// POUs/Controller/Lvl1/OVN (Oven)/FB_OVN
FUNCTION_BLOCK FB_OVN EXTENDS FB_CtrlBase
VAR_INPUT
	/// 0 = Busy, 1 = OFF, 2 = BeltOn, 3 = Manual, 4 = Run, 5 = Error, 6 = Bundverschlusserkennung 
	In_iStatus: INT;
	/// Machine off 
	In_bOff: BOOL;
	/// Band on 
	In_bBeltOn: BOOL;
	/// Manual 
	In_bManual: BOOL;
	/// Standart drying process 
	In_bRun: BOOL;
	/// Resetting error 
	In_bAckError: BOOL;
	/// Actual temperature in deci °C 
	In_adiTemp_dc: ARRAY[0..(MAX_NUMBER_OF_OVEN_MODULES - 1)] OF DINT;
	/// Aactual airflow in % 
	In_adiAir_p: ARRAY[0..(MAX_NUMBER_OF_OVEN_MODULES - 1)] OF DINT;
	/// Actual belt speed in mm/min 
	In_diSpeed_mm_min: DINT;
	/// 1=Information, 2=Warning, 3=Error 
	In_iErrorLevel: INT;
	/// Error ID (e.g. 100=temperature overflow) 
	In_iErrorID: INT;
	In_bDriverConnected: BOOL;
	In_bDriverError: BOOL;
	In_udiDriverErrorID: UDINT;
	In_uliBarcodeNew_1: ULINT;
	In_uliBarcodeNew_2: ULINT;
	In_uiNewElement_1: UINT;
	In_uiNewElement_2: UINT;
	In_uliBarcodeDelete_1: ULINT;
	In_uliBarcodeDelete_2: ULINT;
	In_uiDeleteElement_1: UINT;
	In_uiDeleteElement_2: UINT;
END_VAR
VAR
	/// Specific interface struct for public access
	SIf: T_Ctrl_SIf_OVN;
	/// this allows to detect parameter changes
	lastSifPar: T_Ctrl_SIf_OVN_Par;
	/// pointer to function block
	p_fbIBH: POINTER TO FB_IBH;
	p_fbIBH_CIf: POINTER TO BASE_PLC.T_Ctrl_CIf;
	/// Monitors
	afbTempMonitors: ARRAY[0..(MAX_NUMBER_OF_OVEN_MODULES - 1)] OF FB_MONITOR;
	afbAirMonitors: ARRAY[0..(MAX_NUMBER_OF_OVEN_MODULES - 1)] OF FB_MONITOR;
	fbSpeedMonitor: FB_MONITOR;
	udiTimeInBand: UDINT;
	/// Tracker
	fbTracker: FB_Tracker;
	/// Error Tracking
	iLastCalledAlarmNr: INT;
	uiNewElementOld_1: UINT;
	uiNewElementOld_2: UINT;
	uiDeleteElementOld_1: UINT;
	uiDeleteElementOld_2: UINT;
END_VAR

(*__________________________________________________________________________________________________
¦	
¦	Vistaprint Schweiz GmbH
¦	CH - 8401 Winterthur
¦
¦	www.vistaprint.ch - info@vistaprint.ch
¦___________________________________________________________________________________________________

Function desription:
Oven Controller Implementation

History:
Version		Date			Author		Comment
---------------------------------------------------------------------------------------------------
0.00.1		10.12.2013		BB			Start history
___________________________________________________________________________________________________*)

// check if child pointer valid
IF (me.bolActivate) THEN // cyclic call enabled
	
	IF (CIf.Info.bolInitDone=FALSE) THEN // first cycle -> init
		CtrlInit();
		CIf.Info.bolInitDone := TRUE;
	ELSE
		CycleStartDuty();
		
		Always();
		
		StateMachine();
		
		CycleEndDuty();
	END_IF
	
END_IF;

{attribute 'object_name' := 'Always'}
METHOD PROTECTED Always : BOOL
VAR
	fbOVN: INT;
	bResettable: BOOL;
END_VAR
SUPER^.Always();

// ----------------------------------------------------------------------------------
// cyclic actions outside of statemachine
IF (me.StateMachine.intState<>cSTA_SINGLE_ANSWER) THEN
	
	// copy number of modules to IBH driver
	p_fbIBH^.getCtrlSIf()^.Cfg.uiNumberOfModules := SIf.Cfg.uiNumberOfModules;
	
	// check parameter from GUI
	THIS^.checkParameter();
	
	// write input values directly to SIf.Cur
	SIf.Cur.diSpeed_mm_min := THIS^.In_diSpeed_mm_min;
	SIf.Cur.adiAir_p := THIS^.In_adiAir_p;
	SIf.Cur.adiTemp_dc := THIS^.In_adiTemp_dc;
	
	// remove old elements from Tracker
	IF In_uiDeleteElement_1<>uiDeleteElementOld_1 THEN
		uiDeleteElementOld_1 := In_uiDeleteElement_1;
		fbTracker.deleteElement(In_uliBarcodeDelete_1, SIf.Cfg.bolDataChannelEnable);
	END_IF
	IF In_uiDeleteElement_2<>uiDeleteElementOld_2 THEN
		uiDeleteElementOld_2 := In_uiDeleteElement_2;
		fbTracker.deleteElement(In_uliBarcodeDelete_2, SIf.Cfg.bolDataChannelEnable);
	END_IF
	
	// update Tracker
	fbTracker.update(In_adiTemp_mc:=In_adiTemp_dc, In_diSpeed_mm_min:=In_diSpeed_mm_min,bolSendToSaber:=SIf.Cfg.bolDataChannelEnable);
	
	// add new elements to Tracker
	IF In_uiNewElement_1<>uiNewElementOld_1 THEN
		uiNewElementOld_1 := In_uiNewElement_1;
		fbTracker.addElement(In_uliBarcodeNew_1);
	END_IF
	IF In_uiNewElement_2<>uiNewElementOld_2 THEN
		uiNewElementOld_2 := In_uiNewElement_2;
		fbTracker.addElement(In_uliBarcodeNew_2);
	END_IF
	
	// check errors when higher than PONBusy
	IF (me.StateMachine.intState>=Base_PLC.cSTA_PON) AND (NOT CIf.SwCfg.bolSimulation) THEN
		
		// go to error if Driver connection is lost
		IF 		NOT THIS^.In_bDriverConnected
			AND	me.StateMachine.intState<>Base_PLC.cSTA_ERROR
			AND	me.StateMachine.intState<>Base_PLC.cSTA_ERRORQuit THEN
				pfbAlarmCtrl^.setAlarm(CIf.Info.intCtrlId,INT_TO_UDINT(E_ALM_OVN.ConnectionError),UDINT_TO_DINT(THIS^.In_udiDriverErrorID),ADR(SIf.Alm),E_AlmState.RST,CIf.Job.eMe_ActivAlmClass);
				me.StateMachine.intStateNext := Base_PLC.cSTA_ERROR;
				iLastCalledAlarmNr := E_ALM_OVN.ConnectionError;
		END_IF
		
		// check Tesoma Errors, ErrorLevel 1 (Info) and 2 (Warning) don't exist
		IF THIS^.In_iErrorLevel=3 THEN
			chooseTesomaErrors(bResettable);
			IF 		me.StateMachine.intState<>Base_PLC.cSTA_ERROR
				AND	me.StateMachine.intState<>Base_PLC.cSTA_ERRORQuit
				and me.StateMachine.intStateNext<>Base_PLC.cSTA_ERROR THEN
					me.StateMachine.intStateNext := Base_PLC.cSTA_ERROR;
			END_IF
		END_IF
		
	END_IF
	
END_IF

// ----------------------------------------------------------------------------------
// overrule error always from base -> no EOFF State!! in EOFF go to OFF
IF (me.StateMachine.intStateNext = cSTA_EOFFBusy) THEN
	IF (me.StateMachine.intState = cSTA_OFF) THEN
		me.StateMachine.intStateNext := cSTA_OFF;
	ELSE // stay in OFF
		me.StateMachine.intStateNext := cSTA_OFFBusy;
	END_IF
END_IF
END_METHOD

{attribute 'object_name' := 'checkParameter'}
METHOD checkParameter : BOOL
VAR
	uiIdx: UINT;
END_VAR
// Belt Speed
IF (SIf.Par.diSpeed_mm_min > SIf.Cfg.diMaxSpeed_mm_min) THEN
	pfbAlarmCtrl^.setAlarm(CIf.Info.intCtrlId,INT_TO_UDINT(E_ALM_OVN.ParameterWarning),0,ADR(SIf.Alm),E_AlmState.RST,CIf.Job.eMe_ActivAlmClass);
	SIf.Par.diSpeed_mm_min := SIf.Cfg.diMaxSpeed_mm_min;
ELSIF (SIf.Par.diSpeed_mm_min < SIf.Cfg.diMinSpeed_mm_min) THEN
	pfbAlarmCtrl^.setAlarm(CIf.Info.intCtrlId,INT_TO_UDINT(E_ALM_OVN.ParameterWarning),0,ADR(SIf.Alm),E_AlmState.RST,CIf.Job.eMe_ActivAlmClass);
	SIf.Par.diSpeed_mm_min := SIf.Cfg.diMinSpeed_mm_min;
END_IF

// Temperature
FOR uiIdx:=0 TO SIf.Cfg.uiNumberOfModules-1 BY 1 DO
	IF (SIf.Par.adiTemp_dc[uiIdx] > SIf.Cfg.diMaxTemp_dc) THEN
		pfbAlarmCtrl^.setAlarm(CIf.Info.intCtrlId,INT_TO_UDINT(E_ALM_OVN.ParameterWarning),uiIdx,ADR(SIf.Alm),E_AlmState.RST,CIf.Job.eMe_ActivAlmClass);
		SIf.Par.adiTemp_dc[uiIdx] := SIf.Cfg.diMaxTemp_dc;
	ELSIF (SIf.Par.adiTemp_dc[uiIdx] < SIf.Cfg.diMinTemp_dc) THEN
		pfbAlarmCtrl^.setAlarm(CIf.Info.intCtrlId,INT_TO_UDINT(E_ALM_OVN.ParameterWarning),uiIdx,ADR(SIf.Alm),E_AlmState.RST,CIf.Job.eMe_ActivAlmClass);
		SIf.Par.adiTemp_dc[uiIdx] := SIf.Cfg.diMinTemp_dc;
	END_IF
END_FOR

// Airflow
FOR uiIdx:=0 TO SIf.Cfg.uiNumberOfModules-1 BY 1 DO
	IF (SIf.Par.adiAir_p[uiIdx] > SIf.Cfg.diMaxAir_p) THEN
		pfbAlarmCtrl^.setAlarm(CIf.Info.intCtrlId,INT_TO_UDINT(E_ALM_OVN.ParameterWarning),uiIdx,ADR(SIf.Alm),E_AlmState.RST,CIf.Job.eMe_ActivAlmClass);
		SIf.Par.adiAir_p[uiIdx] := SIf.Cfg.diMaxAir_p;
	ELSIF (SIf.Par.adiAir_p[uiIdx] < SIf.Cfg.diMinAir_p) THEN
		pfbAlarmCtrl^.setAlarm(CIf.Info.intCtrlId,INT_TO_UDINT(E_ALM_OVN.ParameterWarning),uiIdx,ADR(SIf.Alm),E_AlmState.RST,CIf.Job.eMe_ActivAlmClass);
		SIf.Par.adiAir_p[uiIdx] := SIf.Cfg.diMinAir_p;
	END_IF
END_FOR
END_METHOD

{attribute 'object_name' := 'chooseTesomaErrors'}
METHOD chooseTesomaErrors : BOOL
VAR_IN_OUT
	bResettable: BOOL;
END_VAR
bResettable := FALSE;

CASE THIS^.In_iErrorID OF
	// Tesoma10000
	10000:
		bResettable := TRUE;
		pfbAlarmCtrl^.setAlarm(CIf.Info.intCtrlId,INT_TO_UDINT(E_ALM_OVN.Tesoma10000),In_iErrorID,ADR(SIf.Alm),E_AlmState.RST,CIf.Job.eMe_ActivAlmClass);
	// Tesoma10002
	10002:
		pfbAlarmCtrl^.setAlarm(CIf.Info.intCtrlId,INT_TO_UDINT(E_ALM_OVN.Tesoma10002),In_iErrorID,ADR(SIf.Alm),E_AlmState.RST,CIf.Job.eMe_ActivAlmClass);
	// Tesoma10003
	10003:
		pfbAlarmCtrl^.setAlarm(CIf.Info.intCtrlId,INT_TO_UDINT(E_ALM_OVN.Tesoma10003),In_iErrorID,ADR(SIf.Alm),E_AlmState.RST,CIf.Job.eMe_ActivAlmClass);
	// Tesoma10006
	10006:
		pfbAlarmCtrl^.setAlarm(CIf.Info.intCtrlId,INT_TO_UDINT(E_ALM_OVN.Tesoma10006),In_iErrorID,ADR(SIf.Alm),E_AlmState.RST,CIf.Job.eMe_ActivAlmClass);
	// Tesoma10010
	10010:
		bResettable := TRUE;
		pfbAlarmCtrl^.setAlarm(CIf.Info.intCtrlId,INT_TO_UDINT(E_ALM_OVN.Tesoma10010),In_iErrorID,ADR(SIf.Alm),E_AlmState.RST,CIf.Job.eMe_ActivAlmClass);
	// Tesoma10011
	10011:
		bResettable := TRUE;
		pfbAlarmCtrl^.setAlarm(CIf.Info.intCtrlId,INT_TO_UDINT(E_ALM_OVN.Tesoma10011),In_iErrorID,ADR(SIf.Alm),E_AlmState.RST,CIf.Job.eMe_ActivAlmClass);
	// Tesoma10012
	10012:
		bResettable := TRUE;
		pfbAlarmCtrl^.setAlarm(CIf.Info.intCtrlId,INT_TO_UDINT(E_ALM_OVN.Tesoma10012),In_iErrorID,ADR(SIf.Alm),E_AlmState.RST,CIf.Job.eMe_ActivAlmClass);
	// Tesoma10013
	10013:
		pfbAlarmCtrl^.setAlarm(CIf.Info.intCtrlId,INT_TO_UDINT(E_ALM_OVN.Tesoma10013),In_iErrorID,ADR(SIf.Alm),E_AlmState.RST,CIf.Job.eMe_ActivAlmClass);
	// Tesoma10014
	10014:
		bResettable := TRUE;
		pfbAlarmCtrl^.setAlarm(CIf.Info.intCtrlId,INT_TO_UDINT(E_ALM_OVN.Tesoma10014),In_iErrorID,ADR(SIf.Alm),E_AlmState.RST,CIf.Job.eMe_ActivAlmClass);
	// Tesoma10016
	10016:
		pfbAlarmCtrl^.setAlarm(CIf.Info.intCtrlId,INT_TO_UDINT(E_ALM_OVN.Tesoma10016),In_iErrorID,ADR(SIf.Alm),E_AlmState.RST,CIf.Job.eMe_ActivAlmClass);
	// Tesoma10023
	10023:
		pfbAlarmCtrl^.setAlarm(CIf.Info.intCtrlId,INT_TO_UDINT(E_ALM_OVN.Tesoma10023),In_iErrorID,ADR(SIf.Alm),E_AlmState.RST,CIf.Job.eMe_ActivAlmClass);
	// Tesoma10024
	10024:
		pfbAlarmCtrl^.setAlarm(CIf.Info.intCtrlId,INT_TO_UDINT(E_ALM_OVN.Tesoma10024),In_iErrorID,ADR(SIf.Alm),E_AlmState.RST,CIf.Job.eMe_ActivAlmClass);
	// Tesoma10025
	10025:
		pfbAlarmCtrl^.setAlarm(CIf.Info.intCtrlId,INT_TO_UDINT(E_ALM_OVN.Tesoma10025),In_iErrorID,ADR(SIf.Alm),E_AlmState.RST,CIf.Job.eMe_ActivAlmClass);
	// Tesoma10026
	10026:
		pfbAlarmCtrl^.setAlarm(CIf.Info.intCtrlId,INT_TO_UDINT(E_ALM_OVN.Tesoma10026),In_iErrorID,ADR(SIf.Alm),E_AlmState.RST,CIf.Job.eMe_ActivAlmClass);
	// Tesoma10027
	10027:
		pfbAlarmCtrl^.setAlarm(CIf.Info.intCtrlId,INT_TO_UDINT(E_ALM_OVN.Tesoma10027),In_iErrorID,ADR(SIf.Alm),E_AlmState.RST,CIf.Job.eMe_ActivAlmClass);
	// Tesoma10030
	10030:
		pfbAlarmCtrl^.setAlarm(CIf.Info.intCtrlId,INT_TO_UDINT(E_ALM_OVN.Tesoma10030),In_iErrorID,ADR(SIf.Alm),E_AlmState.RST,CIf.Job.eMe_ActivAlmClass);
	// Tesoma10031
	10031:
		pfbAlarmCtrl^.setAlarm(CIf.Info.intCtrlId,INT_TO_UDINT(E_ALM_OVN.Tesoma10031),In_iErrorID,ADR(SIf.Alm),E_AlmState.RST,CIf.Job.eMe_ActivAlmClass);
	// Tesoma10032
	10032:
		pfbAlarmCtrl^.setAlarm(CIf.Info.intCtrlId,INT_TO_UDINT(E_ALM_OVN.Tesoma10032),In_iErrorID,ADR(SIf.Alm),E_AlmState.RST,CIf.Job.eMe_ActivAlmClass);
	// Tesoma10034
	10034:
		pfbAlarmCtrl^.setAlarm(CIf.Info.intCtrlId,INT_TO_UDINT(E_ALM_OVN.Tesoma10034),In_iErrorID,ADR(SIf.Alm),E_AlmState.RST,CIf.Job.eMe_ActivAlmClass);
	// Tesoma10x00
	10100, 10200, 10300, 10400, 10500, 10600, 10700, 10800, 10900:
		bResettable := TRUE;
		pfbAlarmCtrl^.setAlarm(CIf.Info.intCtrlId,INT_TO_UDINT(E_ALM_OVN.Tesoma10x00),In_iErrorID,ADR(SIf.Alm),E_AlmState.RST,CIf.Job.eMe_ActivAlmClass);
	// Tesoma10x01
	10101, 10201, 10301, 10401, 10501, 10601, 10701, 10801, 10901:
		bResettable := TRUE;
		pfbAlarmCtrl^.setAlarm(CIf.Info.intCtrlId,INT_TO_UDINT(E_ALM_OVN.Tesoma10x01),In_iErrorID,ADR(SIf.Alm),E_AlmState.RST,CIf.Job.eMe_ActivAlmClass);
	// Tesoma10x02
	10102, 10202, 10302, 10402, 10502, 10602, 10702, 10802, 10902:
		bResettable := TRUE;
		pfbAlarmCtrl^.setAlarm(CIf.Info.intCtrlId,INT_TO_UDINT(E_ALM_OVN.Tesoma10x02),In_iErrorID,ADR(SIf.Alm),E_AlmState.RST,CIf.Job.eMe_ActivAlmClass);
	// Tesoma10x03
	10103, 10203, 10303, 10403, 10503, 10603, 10703, 10803, 10903:
		bResettable := TRUE;
		pfbAlarmCtrl^.setAlarm(CIf.Info.intCtrlId,INT_TO_UDINT(E_ALM_OVN.Tesoma10x03),In_iErrorID,ADR(SIf.Alm),E_AlmState.RST,CIf.Job.eMe_ActivAlmClass);
	// Tesoma10x07
	10107, 10207, 10307, 10407, 10507, 10607, 10707, 10807, 10907:
		bResettable := TRUE;
		pfbAlarmCtrl^.setAlarm(CIf.Info.intCtrlId,INT_TO_UDINT(E_ALM_OVN.Tesoma10x07),In_iErrorID,ADR(SIf.Alm),E_AlmState.RST,CIf.Job.eMe_ActivAlmClass);
	// Tesoma10x13
	10113, 10213, 10313, 10413, 10513, 10613, 10713, 10813, 10913:
		pfbAlarmCtrl^.setAlarm(CIf.Info.intCtrlId,INT_TO_UDINT(E_ALM_OVN.Tesoma10x13),In_iErrorID,ADR(SIf.Alm),E_AlmState.RST,CIf.Job.eMe_ActivAlmClass);
	// Tesoma10x14
	10114, 10214, 10314, 10414, 10514, 10614, 10714, 10814, 10914:
		pfbAlarmCtrl^.setAlarm(CIf.Info.intCtrlId,INT_TO_UDINT(E_ALM_OVN.Tesoma10x14),In_iErrorID,ADR(SIf.Alm),E_AlmState.RST,CIf.Job.eMe_ActivAlmClass);
	// Tesoma10x15
	10115, 10215, 10315, 10415, 10515, 10615, 10715, 10815, 10915:
		pfbAlarmCtrl^.setAlarm(CIf.Info.intCtrlId,INT_TO_UDINT(E_ALM_OVN.Tesoma10x15),In_iErrorID,ADR(SIf.Alm),E_AlmState.RST,CIf.Job.eMe_ActivAlmClass);
	// Tesoma13x00
	13100, 13200, 13300, 13400, 13500, 13600, 13700, 13800, 13900:
		bResettable := TRUE;
		pfbAlarmCtrl^.setAlarm(CIf.Info.intCtrlId,INT_TO_UDINT(E_ALM_OVN.Tesoma13x00),In_iErrorID,ADR(SIf.Alm),E_AlmState.RST,CIf.Job.eMe_ActivAlmClass);
ELSE
	// TesomaUnknown
		pfbAlarmCtrl^.setAlarm(CIf.Info.intCtrlId,INT_TO_UDINT(E_ALM_OVN.TesomaUnknown),In_iErrorID,ADR(SIf.Alm),E_AlmState.RST,CIf.Job.eMe_ActivAlmClass);
END_CASE
END_METHOD

{attribute 'object_name' := 'CtrlInit'}
METHOD CtrlInit : BOOL
SUPER^.CtrlInit();

// add childs
p_fbIBH_CIf := THIS^.AddChild(p_fbIBH^);

// Tracker Init
fbTracker.numberOfModules := SIf.Cfg.uiNumberOfModules;
fbTracker.sampleTime_us := me.FUBInfo.udiSample_us;
fbTracker.moduleLength_mm := SIf.Cfg.diModuleLength_mm;
fbTracker.distanceBeforeOven_mm := SIf.Cfg.diDistanceBeforeOven_mm;	//TODO: BB: This should be the distance from the barcode reader to the begin of the first module of the oven
fbTracker.distanceAfterOven_mm := SIf.Cfg.diDistanceAfterOven_mm;	//TODO: BB: This should be the distance from the barcode reader to the end of the first module of the oven
END_METHOD

PROPERTY PUBLIC CtrlSIf : POINTER TO T_Ctrl_SIf_OVN
GET
CtrlSIf := ADR(SIf);
END_GET
END_PROPERTY

PROPERTY DataChannel : POINTER TO FB_DataChannelSenderFifo
SET
fbTracker.DataChannel := DataChannel;
END_SET
END_PROPERTY

{attribute 'object_name' := 'FB_init'}
METHOD FB_init : BOOL
VAR_INPUT
	///if TRUE, the retain variables are initialized (warm start / cold start)
	bInitRetains: BOOL;
	///if TRUE, the instance afterwards gets moved into the copy code (online change)
	bInCopyCode: BOOL;
END_VAR
VAR
	uiIdx: UINT;
END_VAR
//------------------------------------------------------------------------------------------------------------------------
// to manually change in new FUB implementation!!!
// define valid commands for this controller
FOR uiIdx:=0 TO (SIZEOF(CIf.Job.aCmdList)/SIZEOF(CIf.Job.aCmdList[0])-1) BY 1 DO
	IF (CIf.Job.aCmdList[uiIdx].intCmd=cSTA_INITIALIZED) THEN
		// found first empty array element
		EXIT;
	END_IF
END_FOR

// Add configuration of own comands
CIf.Job.aCmdList[uiIdx].intCmd := OVN_CmdState.cCMD_BELTONLY;
CIf.Job.aCmdList[uiIdx].strName := 'BELTONLY';
CIf.Job.aCmdList[uiIdx].bolAvailable := TRUE;
uiIdx := uiIdx+1;
CIf.Job.aCmdList[uiIdx].intCmd := Base_PLC.cCMD_RUN;
CIf.Job.aCmdList[uiIdx].strName := 'RUN';
CIf.Job.aCmdList[uiIdx].bolAvailable := TRUE;

// set name of class/typ
CIf.Info.strType := 'FB_OVN';
CIf.Info.strFullName := 'Oven';

// set alarm class
SIf.Alm[E_ALM_OVN.TempError].eAlmClass := E_AlmClass.TSTOP;
SIf.Alm[E_ALM_OVN.TempError].strText := 'Temperature Error';
SIf.Alm[E_ALM_OVN.AirError].eAlmClass := E_AlmClass.TSTOP;
SIf.Alm[E_ALM_OVN.AirError].strText := 'Airflow Error';
SIf.Alm[E_ALM_OVN.SpeedError].eAlmClass := E_AlmClass.TSTOP;
SIf.Alm[E_ALM_OVN.SpeedError].strText := 'Band Speed Error';
SIf.Alm[E_ALM_OVN.TimeoutError].eAlmClass := E_AlmClass.TSTOP;
SIf.Alm[E_ALM_OVN.TimeoutError].strText := 'Timeout Error on State Change';
SIf.Alm[E_ALM_OVN.ParameterWarning].eAlmClass := E_AlmClass.WARNING;
SIf.Alm[E_ALM_OVN.ParameterWarning].strText := 'Parameter Warning - Parameters got adjusted within the allowed limits';
SIf.Alm[E_ALM_OVN.ConnectionError].eAlmClass := E_AlmClass.TSTOP;
SIf.Alm[E_ALM_OVN.ConnectionError].strText := 'Connection Error';
SIf.Alm[E_ALM_OVN.WrongMode].eAlmClass := E_AlmClass.TSTOP;
SIf.Alm[E_ALM_OVN.WrongMode].strText := 'Wrong Mode - Possible Manual Intervention';

SIf.Alm[E_ALM_OVN.Tesoma10000].eAlmClass := E_AlmClass.TSTOP;
SIf.Alm[E_ALM_OVN.Tesoma10000].strText := 'Tesoma - Overtemperature Power Section';
SIf.Alm[E_ALM_OVN.Tesoma10002].eAlmClass := E_AlmClass.TSTOP;
SIf.Alm[E_ALM_OVN.Tesoma10002].strText := 'Tesoma - Failure of Active Cooling Unit';
SIf.Alm[E_ALM_OVN.Tesoma10003].eAlmClass := E_AlmClass.TSTOP;
SIf.Alm[E_ALM_OVN.Tesoma10003].strText := 'Tesoma - Active Cooling Unit not Running';
SIf.Alm[E_ALM_OVN.Tesoma10006].eAlmClass := E_AlmClass.TSTOP;
SIf.Alm[E_ALM_OVN.Tesoma10006].strText := 'Tesoma - Failure Fuse General';
SIf.Alm[E_ALM_OVN.Tesoma10010].eAlmClass := E_AlmClass.TSTOP;
SIf.Alm[E_ALM_OVN.Tesoma10010].strText := 'Tesoma - Belt Position Control Sensor Error';
SIf.Alm[E_ALM_OVN.Tesoma10011].eAlmClass := E_AlmClass.TSTOP;
SIf.Alm[E_ALM_OVN.Tesoma10011].strText := 'Tesoma - Belt Edge Shut Off';
SIf.Alm[E_ALM_OVN.Tesoma10012].eAlmClass := E_AlmClass.TSTOP;
SIf.Alm[E_ALM_OVN.Tesoma10012].strText := 'Tesoma - Fault Belt Speed';
SIf.Alm[E_ALM_OVN.Tesoma10013].eAlmClass := E_AlmClass.TSTOP;
SIf.Alm[E_ALM_OVN.Tesoma10013].strText := 'Tesoma - Transport Overload';
SIf.Alm[E_ALM_OVN.Tesoma10014].eAlmClass := E_AlmClass.TSTOP;
SIf.Alm[E_ALM_OVN.Tesoma10014].strText := 'Tesoma - Belt Control Device Fault';
SIf.Alm[E_ALM_OVN.Tesoma10016].eAlmClass := E_AlmClass.TSTOP;
SIf.Alm[E_ALM_OVN.Tesoma10016].strText := 'Tesoma - Emergency Stop';
SIf.Alm[E_ALM_OVN.Tesoma10023].eAlmClass := E_AlmClass.TSTOP;
SIf.Alm[E_ALM_OVN.Tesoma10023].strText := 'Tesoma - Belt Wear Monitor';
SIf.Alm[E_ALM_OVN.Tesoma10024].eAlmClass := E_AlmClass.TSTOP;
SIf.Alm[E_ALM_OVN.Tesoma10024].strText := 'Tesoma - Control Cabinet Fan';
SIf.Alm[E_ALM_OVN.Tesoma10025].eAlmClass := E_AlmClass.TSTOP;
SIf.Alm[E_ALM_OVN.Tesoma10025].strText := 'Tesoma - Control Cabinet Temperature too High';
SIf.Alm[E_ALM_OVN.Tesoma10026].eAlmClass := E_AlmClass.TSTOP;
SIf.Alm[E_ALM_OVN.Tesoma10026].strText := 'Tesoma - Power Supply Failure';
SIf.Alm[E_ALM_OVN.Tesoma10027].eAlmClass := E_AlmClass.TSTOP;
SIf.Alm[E_ALM_OVN.Tesoma10027].strText := 'Tesoma - Intake Hood Temperature Exceeded';
SIf.Alm[E_ALM_OVN.Tesoma10030].eAlmClass := E_AlmClass.TSTOP;
SIf.Alm[E_ALM_OVN.Tesoma10030].strText := 'Tesoma - Air Pressure too low';
SIf.Alm[E_ALM_OVN.Tesoma10031].eAlmClass := E_AlmClass.TSTOP;
SIf.Alm[E_ALM_OVN.Tesoma10031].strText := 'Tesoma - Belt Position Control not Working';
SIf.Alm[E_ALM_OVN.Tesoma10032].eAlmClass := E_AlmClass.TSTOP;
SIf.Alm[E_ALM_OVN.Tesoma10032].strText := 'Tesoma - Error Cooling Device Control Cabinet';
SIf.Alm[E_ALM_OVN.Tesoma10034].eAlmClass := E_AlmClass.TSTOP;
SIf.Alm[E_ALM_OVN.Tesoma10034].strText := 'Tesoma - Control Cabinet Cooler and Small Drives Fuse Failure';
SIf.Alm[E_ALM_OVN.Tesoma10x00].eAlmClass := E_AlmClass.TSTOP;
SIf.Alm[E_ALM_OVN.Tesoma10x00].strText := 'Tesoma - LimitSwitchingOff';
SIf.Alm[E_ALM_OVN.Tesoma10x01].eAlmClass := E_AlmClass.TSTOP;
SIf.Alm[E_ALM_OVN.Tesoma10x01].strText := 'Tesoma - Overtemperature Safety Temperature Limiter';
SIf.Alm[E_ALM_OVN.Tesoma10x02].eAlmClass := E_AlmClass.TSTOP;
SIf.Alm[E_ALM_OVN.Tesoma10x02].strText := 'Tesoma - Fuse Triggered';
SIf.Alm[E_ALM_OVN.Tesoma10x03].eAlmClass := E_AlmClass.TSTOP;
SIf.Alm[E_ALM_OVN.Tesoma10x03].strText := 'Tesoma - Failure Exhaust Air Differential Pressure Sensor';
SIf.Alm[E_ALM_OVN.Tesoma10x07].eAlmClass := E_AlmClass.TSTOP;
SIf.Alm[E_ALM_OVN.Tesoma10x07].strText := 'Tesoma - Error Frequency Converter';
SIf.Alm[E_ALM_OVN.Tesoma10x13].eAlmClass := E_AlmClass.TSTOP;
SIf.Alm[E_ALM_OVN.Tesoma10x13].strText := 'Tesoma - Temperature Sensor IR Defective';
SIf.Alm[E_ALM_OVN.Tesoma10x14].eAlmClass := E_AlmClass.TSTOP;
SIf.Alm[E_ALM_OVN.Tesoma10x14].strText := 'Tesoma - Fault Frame Cooling System Differential Pressure Sensor';
SIf.Alm[E_ALM_OVN.Tesoma10x15].eAlmClass := E_AlmClass.TSTOP;
SIf.Alm[E_ALM_OVN.Tesoma10x15].strText := 'Tesoma - Fault Exhaust Air Differential Pressure Sensor';
SIf.Alm[E_ALM_OVN.Tesoma13x00].eAlmClass := E_AlmClass.TSTOP;
SIf.Alm[E_ALM_OVN.Tesoma13x00].strText := 'Tesoma - Temperature Fault';
SIf.Alm[E_ALM_OVN.TesomaUnknown].eAlmClass := E_AlmClass.TSTOP;
SIf.Alm[E_ALM_OVN.TesomaUnknown].strText := 'Tesoma - Unknown Error';
SIf.Alm[E_ALM_OVN.HostConnectionLost].eAlmClass := E_AlmClass.TSTOP;
SIf.Alm[E_ALM_OVN.HostConnectionLost].strText := 'Saber Communication Lost';
SIf.Alm[E_ALM_OVN.SettingsChanged].eAlmClass := E_AlmClass.TSTOP;
SIf.Alm[E_ALM_OVN.SettingsChanged].strText := 'Settings Changed';

//*******************************************************************************
// initial values
//*******************************************************************************

// Software configuration
CIf.SwCfg.bolExist := TRUE;
CIf.SwCfg.bolEnable := TRUE;
CIf.SwCfg.bolSimulation := FALSE;

// Configuration
SIf.Cfg.uiNumberOfModules := 4;
SIf.Cfg.diModuleLength_mm := 2000;
SIf.Cfg.diDistanceBeforeOven_mm := 1000;
SIf.Cfg.diDistanceAfterOven_mm := 1000;
SIf.Cfg.diMinAir_p := 40;
SIf.Cfg.diMaxAir_p := 100;
SIf.Cfg.diMaxSpeed_mm_min := 30000;
SIf.Cfg.diMinSpeed_mm_min := 3000;
SIf.Cfg.diMinTemp_dc := 0;
SIf.Cfg.diMaxTemp_dc := 2000;
SIf.Cfg.bAutoContinueAfterConnectionError := FALSE;
SIf.Cfg.bolDataChannelEnable := FALSE;
SIf.Cfg.bIgnoreOffBusyWaitPaper := FALSE;

// Parameter
SIf.Par.diSpeed_mm_min := SIf.Cfg.diMinSpeed_mm_min;
SIf.Par.diSpeedBand1_mm_min := 100;
SIf.Par.diSpeedBand2_mm_min := 200;
SIf.Par.udiSpeedTimeout_ms := 5000;
SIf.Par.udiTimeoutOffBusy_ms := 2000;
SIf.Par.udiTimeoutRunBusyReaction_ms := 1000;
SIf.Par.udiTimeoutRunBusyInBand_ms := 1*60*1000;
SIf.Par.udiTimeoutBeltOnlyReaction_ms := 1000;
SIf.Par.udiTimeoutBeltOnlyBusy_ms := 10000;

FOR uiIdx:=0 TO MAX_NUMBER_OF_OVEN_MODULES-1 BY 1 DO
	SIf.Par.adiTemp_dc[uiIdx] := 1000;
	SIf.Par.adiTempBand1_dc[uiIdx] := 30;
	SIf.Par.adiTempBand2_dc[uiIdx] := 60;
	SIf.Par.audiTempTimeout_ms[uiIdx] := 5000;
	SIf.Par.adiAir_p[uiIdx] := SIf.Cfg.diMinAir_p;
	SIf.Par.adiAirBand1_p[uiIdx] := 2;
	SIf.Par.adiAirBand2_p[uiIdx] := 4;
	SIf.Par.audiAirTimeout_ms[uiIdx] := 5000;
END_FOR
END_METHOD

{attribute 'object_name' := 'getCmdState'}
METHOD PROTECTED getCmdState : STRING
VAR_INPUT
	intCmdState: INT;
	bolState: BOOL;
END_VAR
getCmdState := SUPER^.getCmdState(intCmdState:=intCmdState,bolState:=bolState); // get global/base defined cmds/states

IF (getCmdState='') THEN // global not defined get local
	// get string cmd/state string information in runtime
	IF (bolState=FALSE) THEN
		// cmd's
		CASE intCmdState OF
			OVN_CmdState.cCMD_BELTONLY:
				getCmdState := 'BELTONLY';
		ELSE
			getCmdState := 'Cmd not defined';
		END_CASE;
	ELSE
		// state's
		CASE intCmdState OF
			OVN_CmdState.cSTA_BELTONLY: 
				getCmdState := 'BELTONLY';
			OVN_CmdState.cSTA_BELTONLYbusy: 
				getCmdState := 'BELTONLYbusy';
			OVN_CmdState.cSUB_WAITOFF: 
				getCmdState := 'WAITOFF';
			OVN_CmdState.cSUB_WAITPAPER: 
				getCmdState := 'WAITPAPER';
			OVN_CmdState.cSUB_DONE: 
				getCmdState := 'DONE';
		ELSE
			getCmdState := 'State not defined';
		END_CASE;
	END_IF
END_IF
END_METHOD

{attribute 'object_name' := 'getCtrlSIf'}
METHOD getCtrlSIf : POINTER TO T_Ctrl_SIf_OVN
getCtrlSIf := ADR(SIf);
END_METHOD

PROPERTY IBH : POINTER TO FB_IBH
GET
IBH := p_fbIBH;
END_GET
SET
p_fbIBH := IBH;
END_SET
END_PROPERTY

{attribute 'object_name' := 'sta_BELTONLY'}
METHOD PROTECTED sta_BELTONLY : BOOL
VAR
	uiIdx: UINT;
END_VAR
// state implemetation

// Entry action
//--------------------------------------------------------------------------------------
	IF (me.StateMachine.intState <> me.StateMachine.intStateLastCycle) THEN
		// state changed since last cycle
		me.StateMachine.intStateLastCycle := me.StateMachine.intState;
	END_IF

	
// Cyclic action
//--------------------------------------------------------------------------------------

	// check if parameters have changed
	IF (TC2_SYSTEM.MEMCMP(pBuf1:=ADR(SIf.Par), pBuf2:=ADR(THIS^.lastSifPar), n:=SIZEOF(SIf.Par)) <> 0) THEN
		me.StateMachine.intStateNext := OVN_CmdState.cSTA_BELTONLYBusy;
	END_IF
	
	IF NOT In_bBeltOn OR NOT (In_iStatus=2 OR In_iStatus=6 OR In_iStatus=5) THEN
		pfbAlarmCtrl^.setAlarm(CIf.Info.intCtrlId,INT_TO_UDINT(E_ALM_OVN.WrongMode),0,ADR(SIf.Alm),E_AlmState.RST,CIf.Job.eMe_ActivAlmClass);
		me.StateMachine.intStateNext := Base_PLC.cSTA_ERROR;
	END_IF
	
	// State Change Condition
	IF (me.StateMachine.intStateNext <> Base_PLC.cSTA_ERROR) THEN
		CASE me.intCmd OF
			Base_PLC.cCMD_OFF:
				me.StateMachine.intStateNext := Base_PLC.cSTA_OFFBusy;
		END_CASE
	END_IF


// Exit action
//--------------------------------------------------------------------------------------
	IF (me.StateMachine.intState <> me.StateMachine.intStateNext) THEN
		// state is going to change
		;
	END_IF
END_METHOD

{attribute 'object_name' := 'sta_BELTONLYBusy'}
METHOD PROTECTED sta_BELTONLYBusy : BOOL
VAR
	uiIdx: UINT;
	bReady: BOOL;
	iErrorNumber: INT;
END_VAR
// state implemetation

// Entry action
//--------------------------------------------------------------------------------------
	IF (me.StateMachine.intState <> me.StateMachine.intStateLastCycle) THEN
		// state changed since last cycle
		me.StateMachine.intStateLastCycle := me.StateMachine.intState;
		
		// Set Outputs
		p_fbIBH^.setBeltOn();
		p_fbIBH^.setSpeed(In_diSpeed_mm_min := SIf.Par.diSpeed_mm_min);
		THIS^.lastSifPar := SIf.Par;
	END_IF
	
	
// Cyclic action
//--------------------------------------------------------------------------------------
	
	// check if parameters have changed
	IF (TC2_SYSTEM.MEMCMP(pBuf1:=ADR(SIf.Par), pBuf2:=ADR(THIS^.lastSifPar), n:=SIZEOF(SIf.Par)) <> 0) THEN
		p_fbIBH^.setSpeed(In_diSpeed_mm_min := SIf.Par.diSpeed_mm_min);
		THIS^.lastSifPar := SIf.Par;
	END_IF
	
	// check timeouts
	IF me.StateMachine.udiTimeInState_ms>SIf.Par.udiTimeoutBeltOnlyBusy_ms THEN
		iErrorNumber := 100*me.StateMachine.intState+In_iStatus;
		pfbAlarmCtrl^.setAlarm(CIf.Info.intCtrlId,INT_TO_UDINT(E_ALM_OVN.TimeoutError),iErrorNumber,ADR(SIf.Alm),E_AlmState.RST,CIf.Job.eMe_ActivAlmClass);
		me.StateMachine.intStateNext := Base_PLC.cSTA_ERROR;
	ELSIF me.StateMachine.udiTimeInState_ms>SIf.Par.udiTimeoutBeltOnlyReaction_ms THEN
		IF NOT In_bBeltOn OR NOT ((In_iStatus=2) OR (In_iStatus=6)) THEN
			iErrorNumber := 100*me.StateMachine.intState+In_iStatus;
			pfbAlarmCtrl^.setAlarm(CIf.Info.intCtrlId,INT_TO_UDINT(E_ALM_OVN.TimeoutError),iErrorNumber,ADR(SIf.Alm),E_AlmState.RST,CIf.Job.eMe_ActivAlmClass);
			me.StateMachine.intStateNext := Base_PLC.cSTA_ERROR;
		END_IF
	END_IF
	
	// Check if ready
	bReady := TRUE;
	IF NOT In_bBeltOn OR NOT ((In_iStatus=2) OR (In_iStatus=6)) THEN
		bReady := FALSE;
	END_IF
	IF (ABS(THIS^.In_diSpeed_mm_min - SIf.Par.diSpeed_mm_min) > ABS(SIf.Par.diSpeedBand1_mm_min)) THEN
		bReady := FALSE;
	END_IF
	
	// State Change Condition
	IF (me.StateMachine.intStateNext <> Base_PLC.cSTA_ERROR) THEN
		CASE me.intCmd OF
			// OFF
			Base_PLC.cCMD_OFF:
				me.StateMachine.intStateNext := Base_PLC.cSTA_OFFBusy;
		ELSE
			// DEFAULT
			IF bReady THEN
				me.StateMachine.intStateNext := OVN_CmdState.cSTA_BELTONLY;
			END_IF
		END_CASE
	END_IF


// Exit action
//--------------------------------------------------------------------------------------
	IF (me.StateMachine.intState <> me.StateMachine.intStateNext) THEN
		// state is going to change
		;
	END_IF
END_METHOD

{attribute 'object_name' := 'sta_ERROR'}
METHOD PROTECTED sta_ERROR : BOOL
// state implemetation

// Entry action
//--------------------------------------------------------------------------------------
	IF (me.StateMachine.intState <> me.StateMachine.intStateLastCycle) THEN
		// state changed since last cycle
		me.StateMachine.intStateHistory := me.StateMachine.intStateLastCycle; // -> possibillity to go back to state before error
		me.StateMachine.intStateLastCycle := me.StateMachine.intState;
	END_IF

	
// Cyclic action
//--------------------------------------------------------------------------------------	
	
	// Mark all tracked item as trash
	fbTracker.markAllTrash();
	
	// auto continue after Connection Error
	IF (iLastCalledAlarmNr=E_ALM_OVN.ConnectionError AND SIf.Cfg.bAutoContinueAfterConnectionError) THEN
		IF THIS^.In_bDriverConnected THEN
			CIf.Job.bolAlmReset := TRUE;
			pfbAlarmCtrl^.setAlarm(CIf.Info.intCtrlId,INT_TO_UDINT(E_ALM_OVN.ConnectionError),UDINT_TO_DINT(THIS^.In_udiDriverErrorID),ADR(SIf.Alm),E_AlmState.CLR,CIf.Job.eMe_ActivAlmClass);
		END_IF
	END_IF
	
	// State Change Condition
	IF (CIf.Job.bolAlmReset = TRUE) THEN
		IF (p_fbIBH_CIf^.Job.intState = cSTA_OFF) THEN
			// Start Driver
			p_fbIBH_CIf^.Job.intACmd := IBH_CmdState.cCMD_CONNECT;
		END_IF
		p_fbIBH^.setAckError();
		me.StateMachine.intStateNext := cSTA_ERRORQuit;
	END_IF


// Exit action
//--------------------------------------------------------------------------------------
	IF (me.StateMachine.intState <> me.StateMachine.intStateNext) THEN
		// state is going to change
		;
	END_IF
END_METHOD

{attribute 'object_name' := 'sta_ERRORQuit'}
METHOD PROTECTED sta_ERRORQuit : BOOL
// state implemetation

// Entry action
//--------------------------------------------------------------------------------------
	IF (me.StateMachine.intState <> me.StateMachine.intStateLastCycle) THEN
		// state changed since last cycle
		me.StateMachine.intStateLastCycle := me.StateMachine.intState;
	END_IF

	
// Cyclic action
//--------------------------------------------------------------------------------------	
	
	// State Change Condition
	CASE me.StateMachine.intStateHistory OF
		// RUN
		Base_PLC.cSTA_RUN, Base_PLC.cSTA_RUNBusy:
			me.StateMachine.intStateNext := Base_PLC.cSTA_RUNBusy;
		// PON
		Base_PLC.cSTA_PON, Base_PLC.cSTA_PONBusy:
			me.StateMachine.intStateNext := Base_PLC.cSTA_PONBusy;
		// STOP
		Base_PLC.cSTA_STOP, Base_PLC.cSTA_STOPBusy:
			me.StateMachine.intStateNext := Base_PLC.cSTA_STOPBusy;
		// BELTONLY
		OVN_CmdState.cSTA_BELTONLY, OVN_CmdState.cSTA_BELTONLYBusy:
			me.StateMachine.intStateNext := OVN_CmdState.cSTA_BELTONLYBusy;
	ELSE
		// DEFAULT
		me.StateMachine.intStateNext := Base_PLC.cSTA_OFFBusy;
	END_CASE


// Exit action
//--------------------------------------------------------------------------------------
	IF (me.StateMachine.intState <> me.StateMachine.intStateNext) THEN
		// state is going to change
		
		// Reset iLastCalledAlarmNr
		iLastCalledAlarmNr := E_ALM_OVN.NONE;
	END_IF
END_METHOD

{attribute 'object_name' := 'sta_OFF'}
METHOD PROTECTED sta_OFF : BOOL
VAR
	uiIdx: UINT;
END_VAR
// state implemetation

// Entry action
//--------------------------------------------------------------------------------------
	IF (me.StateMachine.intState <> me.StateMachine.intStateLastCycle) THEN
		// state changed since last cycle
		me.StateMachine.intStateLastCycle := me.StateMachine.intState;
	END_IF

	
// Cyclic action
//--------------------------------------------------------------------------------------
	
	IF NOT In_bOff OR NOT (In_iStatus=1 OR In_iStatus=6 OR In_iStatus=5) THEN
		pfbAlarmCtrl^.setAlarm(CIf.Info.intCtrlId,INT_TO_UDINT(E_ALM_OVN.WrongMode),0,ADR(SIf.Alm),E_AlmState.RST,CIf.Job.eMe_ActivAlmClass);
		me.StateMachine.intStateNext := Base_PLC.cSTA_ERROR;
	END_IF
	
	// State Change Condition
	IF (me.StateMachine.intStateNext <> Base_PLC.cSTA_ERROR) THEN
		CASE me.intCmd OF
			// RUN
			Base_PLC.cCMD_RUN:
				me.StateMachine.intStateNext := Base_PLC.cSTA_RUNBusy;
			// BELTONLY
			OVN_CmdState.cCMD_BELTONLY:
				me.StateMachine.intStateNext := OVN_CmdState.cSTA_BELTONLYBusy;
		ELSE
			// DEFAULT
			;
		END_CASE
	END_IF


// Exit action
//--------------------------------------------------------------------------------------
	IF (me.StateMachine.intState <> me.StateMachine.intStateNext) THEN
		// state is going to change
		;
	END_IF
END_METHOD

{attribute 'object_name' := 'sta_OFFBusy'}
METHOD PROTECTED sta_OFFBusy : BOOL
VAR
	bReady: BOOL;
	iErrorNumber: INT;
	uiIdx: UINT;
	udiCoolDownTime_ms: UDINT;
END_VAR
// state implemetation

// Entry action
//--------------------------------------------------------------------------------------
	IF (me.StateMachine.intState <> me.StateMachine.intStateLastCycle) THEN
		// state changed since last cycle
		me.StateMachine.intStateLastCycle := me.StateMachine.intState;
		me.SubStateMachine.intState 	:= OVN_CmdState.cSUB_WAITOFF;
		me.SubStateMachine.intStateNext := OVN_CmdState.cSUB_WAITOFF;
		
		// Set Outputs
		p_fbIBH^.setOff();
		
		// mark all tracked items as trash
		fbTracker.markAllTrash();
	END_IF

	
// Cyclic action
//--------------------------------------------------------------------------------------
	
	CASE me.SubStateMachine.intState OF
			// WAITOFF
			// ------------------------------------------------------------------------
			OVN_CmdState.cSUB_WAITOFF:
				IF (In_bOff AND ((In_iStatus=1) OR (In_iStatus=6))) THEN
					me.SubStateMachine.intStateNext := OVN_CmdState.cSUB_WAITPAPER;
				ELSIF (me.StateMachine.udiTimeInState_ms>SIf.Par.udiTimeoutOffBusy_ms) THEN
					iErrorNumber := 100*me.StateMachine.intState+In_iStatus;
					pfbAlarmCtrl^.setAlarm(CIf.Info.intCtrlId,INT_TO_UDINT(E_ALM_OVN.TimeoutError),iErrorNumber,ADR(SIf.Alm),E_AlmState.RST,CIf.Job.eMe_ActivAlmClass);
					me.StateMachine.intStateNext := Base_PLC.cSTA_ERROR;
				END_IF
				
			// WAITPAPER
			// ------------------------------------------------------------------------
			OVN_CmdState.cSUB_WAITPAPER:
				udiCoolDownTime_ms := DINT_TO_UDINT((SIf.Cfg.uiNumberOfModules*SIf.Cfg.diModuleLength_mm+SIf.Cfg.diDistanceBeforeOven_mm+SIf.Cfg.diDistanceAfterOven_mm)*60*1000/SIf.Par.diSpeed_mm_min);
				IF (me.StateMachine.udiTimeInState_ms>udiCoolDownTime_ms) OR SIf.Cfg.bIgnoreOffBusyWaitPaper THEN
					me.SubStateMachine.intStateNext := OVN_CmdState.cSUB_DONE;
				END_IF
				
			// DONE
			// ------------------------------------------------------------------------
			OVN_CmdState.cSUB_DONE:
				;
	END_CASE
	
	// State Change Condition
	IF (me.StateMachine.intStateNext <> Base_PLC.cSTA_ERROR) THEN
		CASE me.intCmd OF
			// RUN
			Base_PLC.cCMD_RUN:
				me.StateMachine.intStateNext := Base_PLC.cSTA_RUNBusy;
			// BELTONLY
			OVN_CmdState.cCMD_BELTONLY:
				me.StateMachine.intStateNext := OVN_CmdState.cSTA_BELTONLYBusy;
		ELSE
			// DEFAULT
			IF (me.SubStateMachine.intState=OVN_CmdState.cSUB_DONE) THEN
				me.StateMachine.intStateNext := Base_PLC.cCMD_OFF;
			END_IF
		END_CASE
	END_IF


// Exit action
//--------------------------------------------------------------------------------------
	IF (me.StateMachine.intState <> me.StateMachine.intStateNext) THEN
		// state is going to change
		;
	END_IF
END_METHOD

{attribute 'object_name' := 'sta_PON'}
METHOD PROTECTED sta_PON : BOOL
VAR
	uiIdx: UINT;
END_VAR
// state implemetation

// Entry action
//--------------------------------------------------------------------------------------
	IF (me.StateMachine.intState <> me.StateMachine.intStateLastCycle) THEN
		// state changed since last cycle
		me.StateMachine.intStateLastCycle := me.StateMachine.intState;
	END_IF

	
// Cyclic action
//--------------------------------------------------------------------------------------
	
	// State Change Condition
	IF (me.StateMachine.intStateNext <> Base_PLC.cSTA_ERROR) THEN
		IF me.intCmd>Base_PLC.cCMD_PON THEN
			me.StateMachine.intStateNext := Base_PLC.cSTA_OFFBusy;
		END_IF
	END_IF


// Exit action
//--------------------------------------------------------------------------------------
	IF (me.StateMachine.intState <> me.StateMachine.intStateNext) THEN
		// state is going to change
		;
	END_IF
END_METHOD

{attribute 'object_name' := 'sta_PONBusy'}
METHOD PROTECTED sta_PONBusy : BOOL
VAR
	bReady: BOOL := FALSE;
	uiIdx: UINT;
END_VAR
// state implemetation

// Entry action
//--------------------------------------------------------------------------------------
	IF (me.StateMachine.intState <> me.StateMachine.intStateLastCycle) THEN
		// state changed since last cycle
		me.StateMachine.intStateLastCycle := me.StateMachine.intState;
		
		// Start Driver
		p_fbIBH_CIf^.Job.intACmd := IBH_CmdState.cCMD_CONNECT;
		
		uiNewElementOld_1 := In_uiNewElement_1;
		uiNewElementOld_2 := In_uiNewElement_2;
		uiDeleteElementOld_1 := In_uiDeleteElement_1;
		uiDeleteElementOld_2 := In_uiDeleteElement_2;
	END_IF

	
// Cyclic action
//--------------------------------------------------------------------------------------
	
	IF (p_fbIBH_CIf^.Job.intState = cSTA_OFF) THEN
		// Start Driver
		p_fbIBH_CIf^.Job.intACmd := IBH_CmdState.cCMD_CONNECT;
	END_IF
	
	IF THIS^.In_bDriverError THEN
		pfbAlarmCtrl^.setAlarm(CIf.Info.intCtrlId,INT_TO_UDINT(E_ALM_OVN.ConnectionError),UDINT_TO_DINT(THIS^.In_udiDriverErrorID),ADR(SIf.Alm),E_AlmState.RST,CIf.Job.eMe_ActivAlmClass);
		me.StateMachine.intStateNext := Base_PLC.cSTA_ERROR;
		iLastCalledAlarmNr := E_ALM_OVN.ConnectionError;
	END_IF
	
	// State Change Condition
	IF (me.StateMachine.intStateNext <> Base_PLC.cSTA_ERROR) THEN
		IF (THIS^.In_bDriverConnected) THEN
			me.StateMachine.intStateNext := Base_PLC.cSTA_PON;
		END_IF
	END_IF


// Exit action
//--------------------------------------------------------------------------------------
	IF (me.StateMachine.intState <> me.StateMachine.intStateNext) THEN
		// state is going to change
		;
	END_IF
END_METHOD

{attribute 'object_name' := 'sta_RUN'}
METHOD PROTECTED sta_RUN : BOOL
VAR
	uiIdx: UINT;
	bOutOfBand: BOOL := FALSE;
	bError: BOOL := FALSE;
END_VAR
// state implemetation

// Entry action
//--------------------------------------------------------------------------------------
	IF (me.StateMachine.intState <> me.StateMachine.intStateLastCycle) THEN
		// state changed since last cycle
		me.StateMachine.intStateLastCycle := me.StateMachine.intState;
		THIS^.lastSifPar := SIf.Par;
		
		// reset monitor timeouts
		fbSpeedMonitor.resetTime();
		FOR uiIdx:=0 TO SIf.Cfg.uiNumberOfModules-1 BY 1 DO
			afbTempMonitors[uiIdx].resetTime();
			afbAirMonitors[uiIdx].resetTime();
		END_FOR
	END_IF

	
// Cyclic action
//--------------------------------------------------------------------------------------
	
	// check if parameters have changed
	IF (TC2_SYSTEM.MEMCMP(pBuf1:=ADR(SIf.Par), pBuf2:=ADR(THIS^.lastSifPar), n:=SIZEOF(SIf.Par)) <> 0) THEN
		pfbAlarmCtrl^.setAlarm(CIf.Info.intCtrlId,INT_TO_UDINT(E_ALM_OVN.SettingsChanged),0,ADR(SIf.Alm),E_AlmState.RST,CIf.Job.eMe_ActivAlmClass);
		me.StateMachine.intStateNext := Base_PLC.cSTA_RUNBusy;
	END_IF
	
	IF NOT In_bRun OR NOT (In_iStatus=4 OR In_iStatus=6 OR In_iStatus=5) THEN
		pfbAlarmCtrl^.setAlarm(CIf.Info.intCtrlId,INT_TO_UDINT(E_ALM_OVN.WrongMode),0,ADR(SIf.Alm),E_AlmState.RST,CIf.Job.eMe_ActivAlmClass);
		me.StateMachine.intStateNext := Base_PLC.cSTA_ERROR;
	END_IF
	
	// Update Monitors
	IF (me.StateMachine.intStateNext <> Base_PLC.cSTA_RUNBusy) THEN
		// temperature monitors
		FOR uiIdx:=0 TO SIf.Cfg.uiNumberOfModules-1 BY 1 DO
			afbTempMonitors[uiIdx](	diCurrentValue		:= THIS^.SIf.Cur.adiTemp_dc[uiIdx],
									diTargetValue		:= THIS^.SIf.Par.adiTemp_dc[uiIdx],
									diBand1				:= THIS^.SIf.Par.adiTempBand1_dc[uiIdx],
									diBand2				:= THIS^.SIf.Par.adiTempBand2_dc[uiIdx],
									udiTimeoutBand1_ms	:= THIS^.SIf.Par.audiTempTimeout_ms[uiIdx],
									udiSampleTime_ms	:= me.FUBInfo.udiSample_ms,
									bOutOfBand			=> bOutOfBand,
									bError				=> bError);
			IF (bError = TRUE) THEN
				pfbAlarmCtrl^.setAlarm(CIf.Info.intCtrlId,INT_TO_UDINT(E_ALM_OVN.TempError),uiIdx,ADR(SIf.Alm),E_AlmState.RST,CIf.Job.eMe_ActivAlmClass);
				me.StateMachine.intStateNext := Base_PLC.cSTA_ERROR;
			END_IF
		END_FOR
		// airflow monitors
		FOR uiIdx:=0 TO SIf.Cfg.uiNumberOfModules-1 BY 1 DO
			afbAirMonitors[uiIdx](	diCurrentValue		:= THIS^.SIf.Cur.adiAir_p[uiIdx],
									diTargetValue		:= THIS^.SIf.Par.adiAir_p[uiIdx],
									diBand1				:= THIS^.SIf.Par.adiAirBand1_p[uiIdx],
									diBand2				:= THIS^.SIf.Par.adiAirBand2_p[uiIdx],
									udiTimeoutBand1_ms	:= THIS^.SIf.Par.audiAirTimeout_ms[uiIdx],
									udiSampleTime_ms	:= me.FUBInfo.udiSample_ms,
									bOutOfBand			=> bOutOfBand,
									bError				=> bError);
			IF (bError = TRUE) THEN
				pfbAlarmCtrl^.setAlarm(CIf.Info.intCtrlId,INT_TO_UDINT(E_ALM_OVN.AirError),uiIdx,ADR(SIf.Alm),E_AlmState.RST,CIf.Job.eMe_ActivAlmClass);
				me.StateMachine.intStateNext := Base_PLC.cSTA_ERROR;
			END_IF
		END_FOR
		// band speed monitor
		fbSpeedMonitor(	diCurrentValue		:= THIS^.SIf.Cur.diSpeed_mm_min,
						diTargetValue		:= THIS^.SIf.Par.diSpeed_mm_min,
						diBand1				:= THIS^.SIf.Par.diSpeedBand1_mm_min,
						diBand2				:= THIS^.SIf.Par.diSpeedBand2_mm_min,
						udiTimeoutBand1_ms	:= THIS^.SIf.Par.udiSpeedTimeout_ms,
						udiSampleTime_ms	:= me.FUBInfo.udiSample_ms,
						bOutOfBand			=> bOutOfBand,
						bError				=> bError);
		IF (bError = TRUE) THEN
			pfbAlarmCtrl^.setAlarm(CIf.Info.intCtrlId,INT_TO_UDINT(E_ALM_OVN.SpeedError),0,ADR(SIf.Alm),E_AlmState.RST,CIf.Job.eMe_ActivAlmClass);
			me.StateMachine.intStateNext := Base_PLC.cSTA_ERROR;
		END_IF
	END_IF
	
	// State Change Condition
	IF (me.StateMachine.intStateNext <> Base_PLC.cSTA_ERROR) THEN
		CASE me.intCmd OF
			// OFF
			Base_PLC.cCMD_OFF:
				me.StateMachine.intStateNext := Base_PLC.cSTA_OFFBusy;
			// BELTONLY
			OVN_CmdState.cCMD_BELTONLY:
				me.StateMachine.intStateNext := Base_PLC.cSTA_OFFBusy;
		ELSE
			// DEFAULT
			;
		END_CASE
	END_IF


// Exit action
//--------------------------------------------------------------------------------------
	IF (me.StateMachine.intState <> me.StateMachine.intStateNext) THEN
		// state is going to change
		;
	END_IF
END_METHOD

{attribute 'object_name' := 'sta_RUNBusy'}
METHOD PROTECTED sta_RUNBusy : BOOL
VAR
	iIdx: UINT;
	bReady: BOOL;
	iErrorNumber: INT;
END_VAR
// state implemetation

// Entry action
//--------------------------------------------------------------------------------------
	IF (me.StateMachine.intState <> me.StateMachine.intStateLastCycle) THEN
		// state changed since last cycle
		me.StateMachine.intStateLastCycle := me.StateMachine.intState;
		
		// Set Outputs
		p_fbIBH^.setRun();
		p_fbIBH^.setSpeed(In_diSpeed_mm_min := SIf.Par.diSpeed_mm_min);
		p_fbIBH^.setTemp(In_adiTemp_dc := SIf.Par.adiTemp_dc);
		p_fbIBH^.setAirflow(In_adiAir_p := SIf.Par.adiAir_p);
		THIS^.lastSifPar := SIf.Par;
		
		udiTimeInBand := 0;
		
		// delete all tracked items
		fbTracker.deleteAll();
	END_IF
	
// Cyclic action
//--------------------------------------------------------------------------------------
	
	// check if parameters have changed
	IF (TC2_SYSTEM.MEMCMP(pBuf1:=ADR(SIf.Par), pBuf2:=ADR(THIS^.lastSifPar), n:=SIZEOF(SIf.Par)) <> 0) THEN
		p_fbIBH^.setSpeed(In_diSpeed_mm_min := SIf.Par.diSpeed_mm_min);
		p_fbIBH^.setTemp(In_adiTemp_dc := SIf.Par.adiTemp_dc);
		p_fbIBH^.setAirflow(In_adiAir_p := SIf.Par.adiAir_p);
		THIS^.lastSifPar := SIf.Par;
	END_IF
	
	// check timeouts
	IF me.StateMachine.udiTimeInState_ms>SIf.Par.udiTimeoutRunBusyReaction_ms THEN
		IF NOT In_bRun OR NOT ((In_iStatus=0) OR (In_iStatus=4) OR (In_iStatus=6)) THEN
			iErrorNumber := 100*me.StateMachine.intState+In_iStatus;
			pfbAlarmCtrl^.setAlarm(CIf.Info.intCtrlId,INT_TO_UDINT(E_ALM_OVN.TimeoutError),iErrorNumber,ADR(SIf.Alm),E_AlmState.RST,CIf.Job.eMe_ActivAlmClass);
			me.StateMachine.intStateNext := Base_PLC.cSTA_ERROR;
		END_IF
	END_IF
	
	// Check if ready
	bReady := TRUE;
	IF NOT In_bRun OR NOT (In_iStatus=4) THEN	// ignoring In_iStatus=6 since it's only temporary
		bReady := FALSE;
	END_IF
	IF (ABS(THIS^.In_diSpeed_mm_min - SIf.Par.diSpeed_mm_min) > ABS(SIf.Par.diSpeedBand1_mm_min)) THEN
		bReady := FALSE;
	END_IF
	FOR iIdx:=0 TO SIf.Cfg.uiNumberOfModules-1 BY 1 DO
		// Temperature
		IF (ABS(THIS^.In_adiTemp_dc[iIdx] - SIf.Par.adiTemp_dc[iIdx]) > ABS(THIS^.SIf.Par.adiTempBand1_dc[iIdx])) THEN
			bReady := FALSE;
		END_IF
		// Airflow
		IF (ABS(THIS^.In_adiAir_p[iIdx] - THIS^.SIf.Par.adiAir_p[iIdx]) > ABS(THIS^.SIf.Par.adiAirBand1_p[iIdx])) THEN
			bReady := FALSE;
		END_IF
	END_FOR
	
	IF bReady THEN
		udiTimeInBand := udiTimeInBand + me.FUBInfo.udiSample_ms;
		IF udiTimeInBand < SIf.Par.udiTimeoutRunBusyInBand_ms THEN
			bReady := FALSE;
		END_IF
	ELSE
		udiTimeInBand := 0;
	END_IF
	
	// State Change Condition
	IF (me.StateMachine.intStateNext <> Base_PLC.cSTA_ERROR) THEN
		CASE me.intCmd OF
			// OFF
			Base_PLC.cCMD_OFF:
				me.StateMachine.intStateNext := Base_PLC.cSTA_OFFBusy;
			// BELTONLY
			OVN_CmdState.cCMD_BELTONLY:
				me.StateMachine.intStateNext := Base_PLC.cSTA_OFFBusy;
		ELSE
			// DEFAULT
			IF bReady THEN
				me.StateMachine.intStateNext := Base_PLC.cSTA_RUN;
			END_IF
		END_CASE
	END_IF

		
// Exit action
//--------------------------------------------------------------------------------------
	IF (me.StateMachine.intState <> me.StateMachine.intStateNext) THEN
		// state is going to change
		;
	END_IF
END_METHOD

{attribute 'object_name' := 'StateMachine'}
METHOD PROTECTED StateMachine : BOOL
SUPER^.StateMachine();

// main statemachine of base controller
CASE me.StateMachine.intState OF
	// BELTONLY
    OVN_CmdState.cSTA_BELTONLY: 
        THIS^.sta_BELTONLY();
    OVN_CmdState.cSTA_BELTONLYBusy: 
        THIS^.sta_BELTONLYBusy();
	// RUN
	Base_PLC.cSTA_RUN:
		THIS^.sta_RUN();
	Base_PLC.cSTA_RUNBusy:
		THIS^.sta_RUNBusy();
END_CASE;
END_METHOD

END_FUNCTION_BLOCK

// POUs/Controller/Lvl1/OVN (Oven)/FB_Tracker
FUNCTION_BLOCK FB_Tracker
VAR
	fbList: FB_DLL(In_bDoDataWipe := FALSE);
	udiSampleTime_us: UDINT;
	uiNumberOfModules: UINT;
	diModuleLength_mm: DINT;
	diDistanceBeforeOven_mm: DINT;
	diDistanceAfterOven_mm: DINT;
	pDataChannelFifo: POINTER TO FB_DataChannelSenderFifo;
END_VAR

{attribute 'object_name' := 'addElement'}
METHOD addElement
VAR_INPUT
	In_uliBarcode: ULINT;
END_VAR
VAR
	pData: POINTER TO T_Data;
	uiIdx: UINT;
END_VAR
pData := __NEW(T_Data);
pData^.uliBarcode := In_uliBarcode;
pData^.bTrash := FALSE;
pData^.bBarcodeMissed := FALSE;
pData^.diDistance_um := 0;
FOR uiIdx:=0 TO MAX_NUMBER_OF_OVEN_MODULES-1 BY 1 DO
	pData^.diCyclesInModule[uiIdx] := 0;
	pData^.diSumTemp_mc[uiIdx] := 0;
END_FOR

fbList.addElement(In_uliKey:=In_uliBarcode, In_pData:=pData);
END_METHOD

PROPERTY DataChannel : POINTER TO FB_DataChannelSenderFifo
SET
pDataChannelFifo := DataChannel;
END_SET
END_PROPERTY

{attribute 'object_name' := 'deleteAll'}
METHOD deleteAll
fbList.deleteAll();
END_METHOD

{attribute 'object_name' := 'deleteElement'}
METHOD deleteElement : BOOL
VAR_INPUT
	uliBarcodeOfElement: ULINT;
	bolSendToSaber: BOOL;
END_VAR
VAR
	pDeleteElement: POINTER TO T_Element;
	pData: POINTER TO T_Data;
END_VAR
pDeleteElement := fbList.searchElement(In_uliKey:=uliBarcodeOfElement);

IF (pDeleteElement <> 0) THEN
	
	deleteElement := TRUE;
	pData := fbList.deleteElement(pDeleteElement);

	IF bolSendToSaber THEN
		sendData(pData);
	END_IF

	__DELETE(pData);
ELSE
	deleteElement := FALSE;
END_IF
END_METHOD

PROPERTY distanceAfterOven_mm : DINT
GET
distanceAfterOven_mm := diDistanceAfterOven_mm;
END_GET
SET
diDistanceAfterOven_mm := distanceAfterOven_mm;
END_SET
END_PROPERTY

PROPERTY distanceBeforeOven_mm : DINT
GET
distanceBeforeOven_mm := diDistanceBeforeOven_mm;
END_GET
SET
diDistanceBeforeOven_mm := distanceBeforeOven_mm;
END_SET
END_PROPERTY

{attribute 'object_name' := 'markAllTrash'}
METHOD markAllTrash
VAR
	pCurrentElement: POINTER TO T_Element;
	pCurrentData: POINTER TO T_Data;
	uiIdx: UINT;
END_VAR
pCurrentElement := fbList.firstElement();

WHILE (pCurrentElement <> 0) DO
	pCurrentData := pCurrentElement^.pData;
	pCurrentData^.bTrash := TRUE;
	pCurrentElement := pCurrentElement^.pNextElement;
END_WHILE
END_METHOD

PROPERTY moduleLength_mm : DINT
GET
moduleLength_mm := diModuleLength_mm;
END_GET
SET
diModuleLength_mm := moduleLength_mm;
END_SET
END_PROPERTY

{attribute 'object_name' := 'numberOfElements'}
METHOD numberOfElements : UINT
numberOfElements := fbList.numberOfElements();
END_METHOD

PROPERTY numberOfModules : UINT
GET
numberOfModules := uiNumberOfModules;
END_GET
SET
uiNumberOfModules := numberOfModules;
END_SET
END_PROPERTY

PROPERTY sampleTime_us : UDINT
GET
sampleTime_us := udiSampleTime_us;
END_GET
SET
udiSampleTime_us := sampleTime_us;
END_SET
END_PROPERTY

{attribute 'object_name' := 'sendData'}
METHOD sendData : BOOL
VAR_INPUT
	pData: POINTER TO T_Data;
END_VAR
VAR
	uiIdx: UINT;
	pItem: POINTER TO T_Oven_DCH;
END_VAR
IF pDataChannelFifo <> NULL THEN
	pItem := __NEW(T_Oven_DCH);

	// prepare temperature values
	FOR uiIdx:=0 TO MAX_NUMBER_OF_OVEN_MODULES-1 BY 1 DO
		IF pData^.diCyclesInModule[uiIdx] > 0 THEN
			pItem^.diTemperature_mc[uiIdx] := pData^.diSumTemp_mc[uiIdx]/pData^.diCyclesInModule[uiIdx];
		ELSE
			pItem^.diTemperature_mc[uiIdx] := 0;
		END_IF
	END_FOR

	pItem^.rBaseInfo.bolItemAvailable := TRUE;
	
	IF pData^.bTrash THEN
		pItem^.rBaseInfo.eHealth := E_ItemHealth.Ovn_Temperature;
	ELSE
		pItem^.rBaseInfo.eHealth := E_ItemHealth.Healthy;
	END_IF
	pItem^.bTrash := pData^.bTrash;
	
	pItem^.udiIdentification := pData^.uliBarcode;

	pDataChannelFifo^.Push(pItem);
END_IF
END_METHOD

{attribute 'object_name' := 'update'}
METHOD update
VAR_INPUT
	In_adiTemp_mc: ARRAY[0..(MAX_NUMBER_OF_OVEN_MODULES - 1)] OF DINT;
	In_diSpeed_mm_min: DINT;
	bolSendToSaber: BOOL;
END_VAR
VAR
	pCurrentElement: POINTER TO T_Element;
	pCurrentData: POINTER TO T_Data;
	uiIdx: UINT;
END_VAR
pCurrentElement := fbList.firstElement();

WHILE (pCurrentElement <> 0) DO
	pCurrentData := pCurrentElement^.pData;
	
	// Distance
	pCurrentData^.diDistance_um := pCurrentData^.diDistance_um + In_diSpeed_mm_min*1000/60/1000000*UDINT_TO_DINT(udiSampleTime_us);
	
	IF ( pCurrentData^.diDistance_um < (diDistanceBeforeOven_mm * 1000) ) THEN
		// Before the Oven
		;
	ELSIF (pCurrentData^.diDistance_um > (diDistanceBeforeOven_mm+diDistanceAfterOven_mm+uiNumberOfModules*diModuleLength_mm+1000)*1000) THEN
		// 1m after the Barcode scanners after the Oven
		pCurrentData^.bBarcodeMissed := TRUE;
		deleteElement(uliBarcodeOfElement:=pCurrentData^.uliBarcode,bolSendToSaber:=bolSendToSaber);
	ELSE
		// In the Oven
		FOR uiIdx:=0 TO uiNumberOfModules-1 BY 1 DO
			IF (	(pCurrentData^.diDistance_um >= (diDistanceBeforeOven_mm + uiIdx*diModuleLength_mm)*1000)
				AND (pCurrentData^.diDistance_um < (diDistanceBeforeOven_mm + (uiIdx+1)*diModuleLength_mm)*1000) ) THEN
				pCurrentData^.diCyclesInModule[uiIdx] := pCurrentData^.diCyclesInModule[uiIdx] + 1;
				pCurrentData^.diSumTemp_mc[uiIdx] := pCurrentData^.diSumTemp_mc[uiIdx] + In_adiTemp_mc[uiIdx];
			END_IF
		END_FOR
	END_IF
	
	pCurrentElement := pCurrentElement^.pNextElement;
END_WHILE
END_METHOD

END_FUNCTION_BLOCK

// POUs/Controller/Lvl1/PTA [Paper Transport Alignment]/helper/cycle_Pta
FUNCTION cycle_Pta : BOOL
VAR_INPUT
	pPta: POINTER TO T_PTA;
END_VAR

pPta^.ctrl.fbPta_Umc.In_uinStatus 				:= pPta^.io.In_uinUmc_Status;
pPta^.ctrl.fbPta_Umc.In_intMotorActualSpeed 	:= pPta^.io.In_uinUmc_ActualSpeed;
pPta^.ctrl.fbPta_Umc.In_uinMotorSetSpeed 		:= pPta^.io.In_uinUmc_SetSpeed;
pPta^.ctrl.fbPta_Umc.In_uinIOData				:= pPta^.io.In_uinUmc_IOData1;
pPta^.ctrl.fbPta_Umc.In_uinECATState 			:= pPta^.io.In_uinUmc_ECatState;
pPta^.ctrl.fbPta_Umc.In_strNetId 				:= pPta^.io.In_strUmc_ECatNetId;
pPta^.ctrl.fbPta_Umc.In_uintPort 				:= pPta^.io.In_uinUmc_ECatPort;
pPta^.ctrl.fbPta_Umc();
pPta^.io.Out_uinUmc_SetSpeed 					:= pPta^.ctrl.fbPta_Umc.Out_uinSpeedSetpoint;
pPta^.io.Out_uinUmc_Control 					:= pPta^.ctrl.fbPta_Umc.Out_uinControl;

pPta^.ctrl.fbPta.In_bolBeltEntrySensor		 	:= pPta^.io.In_bolInputSensor;
pPta^.ctrl.fbPta.In_bolBeltExitSensor 			:= pPta^.io.In_bolOutputSensor;
pPta^.ctrl.fbPta();

END_FUNCTION

// POUs/Controller/Lvl1/PTA [Paper Transport Alignment]/helper/init_Pta
FUNCTION init_Pta : BOOL
VAR_INPUT
	pPta			: POINTER TO T_PTA;
	/// instance array of all controller instances
	pCtrlInst		: POINTER TO fb_CtrlBase;
	/// common interface array of all controllers (main use for PLC)
	pCtrlCIf		: POINTER TO T_Ctrl_CIf;
END_VAR

pPta^.ctrl.fbPta_Umc.iniAllCtrlArrays(pCtrlInst,pCtrlCIf,pPta^.id.Pta_Umc);
pPta^.ctrl.fbPta.iniAllCtrlArrays(pCtrlInst,pCtrlCIf,pPta^.id.Pta);
pPta^.ctrl.fbPta.Drive := ADR(pPta^.ctrl.fbPta_Umc);

// PTA is a special type of PTB
pPta^.ctrl.fbPta.CtrlSIf^.Cfg.bolVacuumPresent := FALSE;

END_FUNCTION

// POUs/Controller/Lvl1/PTB [Paper Transport Belt]/helper/cycle_Ptb
FUNCTION cycle_Ptb : BOOL
VAR_INPUT
	pPtb: POINTER TO T_PTB;
END_VAR

pPtb^.ctrl.fbPtb_Umc.In_uinStatus 				:= pPtb^.io.In_uinUmc_Status;
pPtb^.ctrl.fbPtb_Umc.In_intMotorActualSpeed 	:= pPtb^.io.In_uinUmc_ActualSpeed;
pPtb^.ctrl.fbPtb_Umc.In_uinMotorSetSpeed 		:= pPtb^.io.In_uinUmc_SetSpeed;
pPtb^.ctrl.fbPtb_Umc.In_uinIOData				:= pPtb^.io.In_uinUmc_IOData1;
pPtb^.ctrl.fbPtb_Umc.In_uinECATState 			:= pPtb^.io.In_uinUmc_ECatState;
pPtb^.ctrl.fbPtb_Umc.In_strNetId 				:= pPtb^.io.In_strUmc_ECatNetId;
pPtb^.ctrl.fbPtb_Umc.In_uintPort 				:= pPtb^.io.In_uinUmc_ECatPort;
pPtb^.ctrl.fbPtb_Umc();
pPtb^.io.Out_uinUmc_SetSpeed 					:= pPtb^.ctrl.fbPtb_Umc.Out_uinSpeedSetpoint;
pPtb^.io.Out_uinUmc_Control 					:= pPtb^.ctrl.fbPtb_Umc.Out_uinControl;

pPtb^.ctrl.fbPtb_Vpc.In_bolPumpOk 				:= pPtb^.io.In_bolVpc_PumpOk;
pPtb^.ctrl.fbPtb_Vpc.In_bolVacuumOk 			:= pPtb^.io.In_bolVpc_VacuumSensor;
pPtb^.ctrl.fbPtb_Vpc();
pPtb^.io.Out_bolVpc_PumpOn 						:= pPtb^.ctrl.fbPtb_Vpc.Out_bolVaccumPumpOn;

pPtb^.ctrl.fbPtb.In_bolBeltEntrySensor		 	:= pPtb^.io.In_bolInputSensor;
pPtb^.ctrl.fbPtb.In_bolBeltExitSensor 			:= pPtb^.io.In_bolOutputSensor;
pPtb^.ctrl.fbPtb();

END_FUNCTION

// POUs/Controller/Lvl1/PTB [Paper Transport Belt]/helper/init_Ptb
FUNCTION init_Ptb : BOOL
VAR_INPUT
	pPtb			: POINTER TO T_PTB;
	/// instance array of all controller instances
	pCtrlInst		: POINTER TO fb_CtrlBase;
	/// common interface array of all controllers (main use for PLC)
	pCtrlCIf		: POINTER TO T_Ctrl_CIf;
END_VAR

pPtb^.ctrl.fbPtb_Vpc.iniAllCtrlArrays(pCtrlInst,pCtrlCIf,pPtb^.id.Ptb_Vpc);
pPtb^.ctrl.fbPtb_Umc.iniAllCtrlArrays(pCtrlInst,pCtrlCIf,pPtb^.id.Ptb_Umc);
pPtb^.ctrl.fbPtb.iniAllCtrlArrays(pCtrlInst,pCtrlCIf,pPtb^.id.Ptb);
pPtb^.ctrl.fbPtb.Drive := ADR(pPtb^.ctrl.fbPtb_Umc);
pPtb^.ctrl.fbPtb.VacuumPump := ADR(pPtb^.ctrl.fbPtb_Vpc);

END_FUNCTION

// POUs/Controller/Lvl1/PTB [Paper Transport Belt]/FB_PTB
FUNCTION_BLOCK FB_PTB EXTENDS FB_CtrlBase
VAR_INPUT
	In_bolBeltEntrySensor		: BOOL;
	In_bolBeltExitSensor		: BOOL;
END_VAR
VAR_OUTPUT
END_VAR
VAR
	/// Specific interface struct for public access
	SIf					: T_Ctrl_SIf_PTB;
	///pointer to function block
	p_fbMotor				: POINTER TO FB_UMC;
	pMotorCIf				: POINTER TO T_Ctrl_CIf;
	p_fbPump				: POINTER TO FB_VPC;
	pPumpCIf				: POINTER TO T_Ctrl_CIf;
	fbEntrySensorDebounce	: FB_PRS;
	fbExitSensorDebounce	: FB_PRS;
	arMotorDirection		: ARRAY [0..E_BELT_DIRECTION.MAX_E_BELT_DIRECTION-1] OF E_TURN_DIRECTION;
	
	// Paper Position Service
	fbPositionService		: FB_PTR;
	udiIdCounter			: UDINT;
	
	// Paper Edge Detectors
	fbPaperEntryPEdge					: TC2_STANDARD.R_TRIG;
	fbPaperEntryNEdge					: TC2_STANDARD.F_TRIG;
	fbPaperExitPEdge					: TC2_STANDARD.R_TRIG;
	fbPaperExitNEdge					: TC2_STANDARD.F_TRIG;
	
END_VAR

(*__________________________________________________________________________________________________
¦	
¦	Vistaprint Schweiz GmbH
¦	CH - 8401 Winterthur
¦
¦	www.vistaprint.ch - info@vistaprint.ch
¦___________________________________________________________________________________________________

Function desription:
Vacuum Pump implementation. 


History:
Version		Date			Author		Comment
---------------------------------------------------------------------------------------------------
0.00.1		09.07.2013		PC			Start history
0.00.2		14.02.2014		AVME/MRU	Cyclic call of fbPositionService added
0.00.3		24.02.2014		AVME/MRU	sta_OFFBusy reworked
0.00.4		02.10.2014		AVME/MRU	Alwaysw reworked for Single_Answer
___________________________________________________________________________________________________*)


SUPER^();

(*
IF (me.bolActivate) THEN // cyclic call enabled
	IF (CIf.Info.bolInitDone=FALSE) THEN // first cycle -> init
		CtrlInit();
		CIf.Info.bolInitDone := TRUE;
	ELSE
		CycleStartDuty();
	
		Always();
		
		StateMachine();
		
		CycleEndDuty();
	END_IF
END_IF;
*)

METHOD PROTECTED Always : BOOL
SUPER^.Always();

// ----------------------------------------------------------------------------------
// cyclic actions outside of statemachine
IF (me.StateMachine.intState<>cSTA_SINGLE_ANSWER) THEN
	
	; // always error supervision
	
END_IF

// ----------------------------------------------------------------------------------
// Conditions Always
IF (((me.Alarm.eActivAlmClass=E_AlmClass.EOFF) OR (me.Alarm.eActivAlmClass=E_AlmClass.OFF) OR (me.intCmd=cCMD_OFF))
		 AND (me.StateMachine.intState<>cSTA_ERROR) AND (me.StateMachine.intState<>cSTA_ERRORQuit) AND
		(me.StateMachine.intState<>cSTA_OFF) AND (me.StateMachine.intState<>cSTA_OFFBusy) AND (me.StateMachine.intState<>cSTA_SINGLE_ANSWER)) THEN
	// alarm evt EOFF, OFF or cmd off
	me.StateMachine.intStateNext := cSTA_OFFBusy;
END_IF

// ----------------------------------------------------------------------------------
// Conditions Always
// overrule error always from base -> no EOFF State!! in EOFF go to OFF
IF (me.StateMachine.intStateNext = cSTA_EOFFBusy) THEN
	IF (me.StateMachine.intState=cSTA_OFF) THEN
		me.StateMachine.intStateNext := cSTA_OFF;
	ELSE // stay in OFF
		me.StateMachine.intStateNext := cSTA_OFFBusy;
	END_IF
END_IF

// -----------------------------------------------------------------------------------
PaperPositionHandling();
// -----------------------------------------------------------------------------------
END_METHOD

METHOD PROTECTED CalculateBeltParameter : UINT
VAR_INPUT
	uinBeltSpeed_mms		: UINT;   	// Belt speed in mm/sec
	reaRpmDistance			: REAL;		// mm/rotation
	pCur		: POINTER TO T_Belt_Cur_Base;
END_VAR
pCur^.uinBeltSpeed_mms := uinBeltSpeed_mms;
// RPM = Speed [mm/sec] / Dispance per Rotation [mm/rpm]
pCur^.uinBeltSpeed_rpm := REAL_TO_UINT(UINT_TO_REAL(uinBeltSpeed_mms) * 60.0 / reaRpmDistance);

CalculateBeltParameter := pCur^.uinBeltSpeed_rpm;
END_METHOD

METHOD PROTECTED CalculateModeParameter : BOOL
VAR_INPUT
END_VAR
CASE SIf.Cfg.eMode OF  
	E_PTB_MODE.ToDistance:
		SIf.Cur.udiTimeToMove_ms		:= REAL_TO_UDINT( 1000.0 * UDINT_TO_REAL(SIf.Par.udiDistanceToMove_mm) / UINT_TO_REAL(SIf.Par.rBeltParam.uinBeltSpeed));
		SIf.Cur.udiTimeToMove_ms		:= SIf.Cur.udiTimeToMove_ms + p_fbMotor^.CtrlSIf^.Par.udiMoveStartLatency - p_fbMotor^.CtrlSIf^.Par.udiMoveStopLatency;
		SIf.Cur.udiDistanceToMove_mm	:= SIf.Par.udiDistanceToMove_mm;
	E_PTB_MODE.ToTime:
		SIf.Cur.udiTimeToMove_ms		:= SIf.Par.udiTimeToMove_ms;
		SIf.Cur.udiDistanceToMove_mm	:= SIf.Par.udiTimeToMove_ms * UINT_TO_UDINT(SIf.Par.rBeltParam.uinBeltSpeed) / 1000;
		SIf.Cur.udiTimeToMove_ms		:= SIf.Cur.udiTimeToMove_ms + p_fbMotor^.CtrlSIf^.Par.udiMoveStartLatency - p_fbMotor^.CtrlSIf^.Par.udiMoveStopLatency;
ELSE
	SIf.Cur.udiTimeToMove_ms		:= 0;
	SIf.Cur.udiDistanceToMove_mm	:= 0;
END_CASE
END_METHOD

METHOD PROTECTED CheckPumpState : BOOL
VAR_INPUT
	intState		: INT;
END_VAR
CheckPumpState := TRUE;

IF SIf.Cfg.bolVacuumPresent THEN
	CheckPumpState := p_fbPump^.CtrlCIf^.Job.intState = intState;
END_IF
END_METHOD

ACTION cmd_OFF:
p_fbMotor^.CtrlCIf^.Job.intACmd := BASE_PLC.cCMD_OFF;
SetPumpComand(cCMD_OFF);
END_ACTION

METHOD PROTECTED cmd_RUN : BOOL
VAR_INPUT
	uinBeltSpeed			: UINT;
END_VAR
SIf.Cur.eActualDirection := SIf.Par.intDirection;
SIf.Cur.rBeltParam.uinBeltSpeed_rpm := CalculateBeltParameter(
											uinBeltSpeed,
											sif.Cfg.rBeltParam.reaRpmDistance_mm,
											ADR(SIf.Cur.rBeltParam));
CalculateModeParameter();
p_fbMotor^.CtrlSIf^.Par.eRotationDirection 	:= THIS^.arMotorDirection[SIf.Par.intDirection];
p_fbMotor^.CtrlSIf^.Par.uinSpeed_rpm 		:= SIf.Cur.rBeltParam.uinBeltSpeed_rpm;
p_fbMotor^.CtrlCIf^.Job.intACmd :=BASE_PLC.cCMD_RUN;
SetPumpComand(cCMD_RUN);
END_METHOD

ACTION cmd_STOP:
p_fbMotor^.CtrlCIf^.Job.intACmd := BASE_PLC.cCMD_STOP;
SetPumpComand(cCMD_RUN);
END_ACTION

METHOD PUBLIC CtrlInit : BOOL
VAR_INPUT
END_VAR
SUPER^.CtrlInit();

pMotorCIf := p_fbMotor^.CtrlCIf;
AddChild(p_fbMotor^);

IF SIf.Cfg.bolVacuumPresent THEN
	pPumpCIf  := p_fbPump^.CtrlCIf;
	AddChild(p_fbPump^);
END_IF

arMotorDirection[E_BELT_DIRECTION.BACKWARD] := SIf.Cfg.rBeltParam.intBackwardDirection;
arMotorDirection[E_BELT_DIRECTION.FORWARD] := SIf.Cfg.rBeltParam.intForwardDirection;

fbPositionService.TimeBase := me.FUBInfo.udiSample_us;
fbPositionService.BeltLength := UDINT_TO_DINT(SIf.Par.udiBeltLength_mm);

CASE SIf.Par.ePaperOrientation OF
	E_PTB_PaperDirection.Portrait:
		fbPositionService.PaperEntryOffset := UINT_TO_INT(SIf.Par.uinPaperHight_mm); 
	E_PTB_PaperDirection.Landscape:
		fbPositionService.PaperEntryOffset := UINT_TO_INT(SIf.Par.uinPaperWidth_mm); 
END_CASE

SIf.Cur.pPositionList := fbPositionService.PositionList;
udiIdCounter := 0;
END_METHOD

PROPERTY PUBLIC CtrlSIf : POINTER TO T_Ctrl_SIf_PTB
GET
CtrlSIf := ADR(SIf);
END_GET
END_PROPERTY

PROPERTY PUBLIC Drive :  POINTER TO FB_UMC
GET
Drive := p_fbMotor;
END_GET
SET
p_fbMotor := Drive;
END_SET
END_PROPERTY

METHOD FB_init : BOOL
VAR_INPUT
	bInitRetains : BOOL; // if TRUE, the retain variables are initialized (warm start / cold start)
	bInCopyCode : BOOL;  // if TRUE, the instance afterwards gets moved into the copy code (online change)
END_VAR
VAR
	iIdx		: UINT;
	iLength		: UINT;	
END_VAR
//------------------------------------------------------------------------------------------------------------------------
// to manually change in new FUB implementation!!!
// define valid commands for this controller
iLength := SIZEOF(CIf.Job.aCmdList)/SIZEOF(CIf.Job.aCmdList[0]);
iIdx := 0;

WHILE (iIdx < iLength) AND (CIf.Job.aCmdList[iIdx].intCmd <> cCMD_INITIALIZED) DO
	iIdx := iIdx + 1; 
END_WHILE

IF (iIdx < iLength) THEN
// Add configuration of own comands	
	CIf.Job.aCmdList[iIdx].intCmd := BASE_PLC.cCMD_RUN;
	CIf.Job.aCmdList[iIdx].strName := 'Run'; 
	CIf.Job.aCmdList[iIdx].bolAvailable := TRUE;
	iIdx := iIdx + 1;
	CIf.Job.aCmdList[iIdx].intCmd := BASE_PLC.cCMD_STOP;
	CIf.Job.aCmdList[iIdx].strName := 'Stop'; 
	CIf.Job.aCmdList[iIdx].bolAvailable := TRUE;
	iIdx := iIdx + 1;
	CIf.Job.aCmdList[iIdx].intCmd := PTB_CmdState.cCMD_EJECTPAPER;
	CIf.Job.aCmdList[iIdx].strName := 'EJECTPAPER'; 
	CIf.Job.aCmdList[iIdx].bolAvailable := TRUE;
	iIdx := iIdx + 1;
	CIf.Job.aCmdList[iIdx].intCmd := PTB_CmdState.cCMD_STACKPAPER;
	CIf.Job.aCmdList[iIdx].strName := 'STACKPAPER'; 
	CIf.Job.aCmdList[iIdx].bolAvailable := TRUE;
ELSE
	// Error if the aCmdList Array is to small
END_IF

// set name of class/typ
CIf.Info.strType := 'FB_PTB';
CIf.Info.strFullName := 'Paper Transport Belt';

// set alarm class
SIf.Alm[E_ALM_PTB.TestAlarm].eAlmClass := Base_PLC.E_AlmClass.TSTOP;
SIf.Alm[E_ALM_PTB.TestAlarm].strText := 'Baum' ;


//*******************************************************************************
// initial values
//*******************************************************************************

// software configuration
CIf.SwCfg.bolExist := TRUE;
CIf.SwCfg.bolEnable := TRUE;
CIf.SwCfg.bolSimulation := FALSE;

// configuration
SIf.Cfg.rBeltParam.intBackwardDirection		:= E_TURN_DIRECTION.LEFT;
SIf.Cfg.rBeltParam.intForwardDirection		:= E_TURN_DIRECTION.RIGHT;
SIf.Cfg.bolVacuumPresent					:= TRUE;
SIf.Cfg.eMode								:= E_PTB_MODE.Endless;
SIf.Cfg.rBeltParam.reaRpmDistance_mm		:= 20.3;

// parameter
SIf.Par.intDirection				:= E_BELT_DIRECTION.FORWARD;
SIf.Par.rBeltParam.uinBeltSpeed		:= 412;
SIf.Par.udiDistanceToMove_mm		:= 0;
SIf.Par.udiTimeToMove_ms			:= 0;
SIf.Par.ePaperOrientation			:= E_PTB_PaperDirection.Portrait;
SIf.Par.uinPaperHight_mm			:= 460;
SIf.Par.uinPaperWidth_mm			:= 320;
SIf.Par.uinInputSignalDebounceTime_ms := 50;


fbEntrySensorDebounce.CtrlSIf^.Par.udiDebounceAbsentTime_ms := SIf.Par.uinInputSignalDebounceTime_ms;
fbEntrySensorDebounce.CtrlSIf^.Par.udiDebouncePresentTime_ms := SIf.Par.uinInputSignalDebounceTime_ms;
fbExitSensorDebounce.CtrlSIf^.Par.udiDebounceAbsentTime_ms := SIf.Par.uinInputSignalDebounceTime_ms;
fbExitSensorDebounce.CtrlSIf^.Par.udiDebouncePresentTime_ms := SIf.Par.uinInputSignalDebounceTime_ms;
END_METHOD

METHOD PROTECTED getCmdState : STRING

VAR_INPUT
	intCmdState: INT;
	bolState: BOOL;
END_VAR
getCmdState := SUPER^.getCmdState(intCmdState:=intCmdState,bolState:=bolState); // get global/base defined cmds/states

IF (getCmdState='') THEN // global not defined get local
	// get string cmd/state string information in runtime
	IF (bolState=FALSE) THEN
		CASE intCmdState OF
			PTB_CmdState.cCMD_EJECTPAPER: 
				getCmdState := 'EJECTPAPER';
			PTB_CmdState.cCMD_STACKPAPER: 
				getCmdState := 'STACKPAPER';
		END_CASE;
	ELSE
		// States's
		CASE intCmdState OF
			PTB_CmdState.cSTA_EJECTPAPER: 
				getCmdState := 'EJECTPAPER';
			PTB_CmdState.cSTA_EJECTPAPERbusy: 
				getCmdState := 'EJECTPAPERbusy';
			PTB_CmdState.cSTA_STACKPAPER: 
				getCmdState := 'STACKPAPER';
			PTB_CmdState.cSTA_STACKPAPERbusy: 
				getCmdState := 'STACKPAPERbusy';
			PTB_CmdState.cSUB_EMPTYstart: 
				getCmdState := 'EMPTYstart';
			PTB_CmdState.cSUB_EMPTYWAITPAPERbusy: 
				getCmdState := 'EMPTYWAITPAPERbusy';
			PTB_CmdState.cSUB_EMPTYWAITPAPERGONEbusy: 
				getCmdState := 'EMPTYWAITPAPERGONEbusy';
			PTB_CmdState.cSUB_PAPERDISTANCEbusy: 
				getCmdState := 'PAPERDISTANCEbusy';
			PTB_CmdState.cSUB_PAPERDISTANCEstart: 
				getCmdState := 'PAPERDISTANCEstart';
			PTB_CmdState.cSUB_STARTENTRYDRIVE: 
				getCmdState := 'STARTENTRYDRIVE';
			PTB_CmdState.cSUB_STARTENTRYDRIVEbusy: 
				getCmdState := 'STARTENTRYDRIVEbusy';
			PTB_CmdState.cSUB_STARTSTACKDELAY: 
				getCmdState := 'STARTSTACKDELAY';
			PTB_CmdState.cSUB_WAITPAPER: 
				getCmdState := 'WAITPAPER';
			PTB_CmdState.cSUB_PAPERDISTANCESTOPbusy:
				getCmdState := 'PAPERDISTANCESTOPbusy';
		END_CASE;
	END_IF
END_IF
END_METHOD

METHOD getCtrlSIf : POINTER TO T_Ctrl_SIf_PTB
getCtrlSIf := ADR(SIf);
END_METHOD

METHOD PROTECTED IoInBridge : BOOL
// digitale and analoge inputs read from hardware or forcing
IF SIf.Cfg.bolExitSensorDebounceEnable THEN
	fbExitSensorDebounce.In_bolPresent := THIS^.In_bolBeltExitSensor;
	fbExitSensorDebounce();
	SIf.In.bolBeltExitSensor.map := fbExitSensorDebounce.Out_bolPresent;
ELSE
	SIf.In.bolBeltExitSensor.map := THIS^.In_bolBeltExitSensor;
END_IF

IF SIf.Cfg.bolEntrySensorDebounceEnable THEN
	fbEntrySensorDebounce.In_bolPresent := THIS^.In_bolBeltExitSensor;
	fbEntrySensorDebounce();
	SIf.In.bolBeltExitSensor.map := fbEntrySensorDebounce.Out_bolPresent;
ELSE
	SIf.In.bolBeltEntrySensor.map := THIS^.In_bolBeltEntrySensor;
END_IF


// Insert also an edge detection
fbPaperEntryPEdge.CLK := SIf.In.bolBeltEntrySensor.map;
fbPaperEntryPEdge();
SIf.In.bolBeltEntrySensorPEdge.map := fbPaperEntryPEdge.Q;

fbPaperEntryNEdge.CLK := SIf.In.bolBeltEntrySensor.map;
fbPaperEntryNEdge();
SIf.In.bolBeltEntrySensorNEdge.map := fbPaperEntryNEdge.Q;

fbPaperExitPEdge.CLK := SIf.In.bolBeltExitSensor.map;
fbPaperExitPEdge();
SIf.In.bolBeltExitSensorPEdge.map := fbPaperExitPEdge.Q;

fbPaperExitNEdge.CLK := SIf.In.bolBeltExitSensor.map;
fbPaperExitNEdge();
SIf.In.bolBeltExitSensorNEdge.map := fbPaperExitNEdge.Q;

IF (CIf.SwCfg.bolSimulation = FALSE) THEN
	getInBol(CIf.Job.bolIoForce,ADR(SIf.In.bolBeltExitSensor));
	getInBol(CIf.Job.bolIoForce,ADR(SIf.In.bolBeltEntrySensor));
	getInBol(CIf.Job.bolIoForce,ADR(SIf.In.bolBeltEntrySensorPEdge));
	getInBol(CIf.Job.bolIoForce,ADR(SIf.In.bolBeltEntrySensorNEdge));
	getInBol(CIf.Job.bolIoForce,ADR(SIf.In.bolBeltExitSensorPEdge));
	getInBol(CIf.Job.bolIoForce,ADR(SIf.In.bolBeltExitSensorNEdge));
ELSE
;	//simulation of global IO
END_IF
END_METHOD

METHOD PROTECTED IoOutBridge : BOOL
VAR
	bolSwitchValvesOff: BOOL;
END_VAR
// digitale and analoge inputs read from hardware or forcing
IF (CIf.SwCfg.bolSimulation = FALSE) THEN
//	setOutBol(CIf.Job.bolIoForce ,ADR(SIf.Out.intActualPosition));
;
//	THIS^.Out_intActualPosition := SIf.Out.intActualPosition.map;
END_IF
END_METHOD

METHOD PROTECTED PaperPositionHandling : BOOL
VAR_INPUT
END_VAR
// Paper Tracking Service
// -----------------------------------------------------------------------------------
CASE me.StateMachine.intState OF
	BASE_PLC.cSTA_RUN:
		fbPositionService.In_uinBeltSpeed := sif.Cur.rBeltParam.uinBeltSpeed_mms;
ELSE
	fbPositionService.In_uinBeltSpeed := 0;
END_CASE

IF SIf.In.bolBeltEntrySensorPEdge.intern THEN
	udiIdCounter := udiIdCounter + 1;
	fbPositionService.Push(udiIdCounter);
END_IF

IF SIf.In.bolBeltEntrySensorNEdge.intern THEN
	fbPositionService.EnterComplete();
END_IF

IF SIf.In.bolBeltExitSensorPEdge.intern THEN
	fbPositionService.Pop();
END_IF

// Cyclic call
fbPositionService();
SIf.Cur.uinPaperOnBelt := fbPositionService.PaperOnBelt;
END_METHOD

PROPERTY PUBLIC PositionList : POINTER TO T_PTR_STRUCT
GET
END_GET
SET
END_SET
END_PROPERTY

METHOD PROTECTED SetPumpComand : BOOL
VAR_INPUT
	intComand		: INT;
END_VAR
SetPumpComand := TRUE;

IF SIf.Cfg.bolVacuumPresent THEN
	p_fbPump^.CtrlCIf^.Job.intACmd := intComand;
END_IF
END_METHOD

METHOD PROTECTED sta_EJECTPAPER : Bool
VAR
	iDifference 		: INT;
END_VAR
// state implemetation
//--------------------------------------------------------------------------------------
// Entry action
	IF (me.StateMachine.intState<>me.StateMachine.intStateLastCycle) THEN
		me.StateMachine.intStateLastCycle := me.StateMachine.intState;
	END_IF


//--------------------------------------------------------------------------------------
// Cyclic action
	IF (me.StateMachine.intState = me.StateMachine.intStateLastCycle) THEN
		CASE me.intCmd OF
			BASE_PLC.cCMD_RUN:
				me.StateMachine.intStateNext := BASE_PLC.cSTA_RUNBusy;
			BASE_PLC.cCMD_STOP:
				me.StateMachine.intStateNext := BASE_PLC.cSTA_STOPBusy;
			PTB_CmdState.cCMD_EJECTPAPER:
				me.StateMachine.intStateNext := PTB_CmdState.cSTA_EJECTPAPERbusy;
			PTB_CmdState.cCMD_STACKPAPER:
				me.StateMachine.intStateNext := PTB_CmdState.cSTA_STACKPAPERbusy;
		END_CASE
	END_IF

//--------------------------------------------------------------------------------------
// Exit action
	IF (me.StateMachine.intState<>me.StateMachine.intStateNext) THEN
		;
	END_IF
END_METHOD

METHOD PROTECTED sta_EJECTPAPERbusy : BOOL
VAR_INPUT
END_VAR
// state implemetation
//--------------------------------------------------------------------------------------
// Entry action
	IF (me.StateMachine.intState<>me.StateMachine.intStateLastCycle) THEN
		me.StateMachine.intStateLastCycle := me.StateMachine.intState;
		cmd_RUN(sif.Par.rBeltParam.uinBeltSpeed);
		me.SubStateMachine.intStateNext := PTB_CmdState.cSUB_EMPTYWAITPAPERbusy;
	END_IF


//--------------------------------------------------------------------------------------
// Cyclic action
	IF (me.StateMachine.intState=me.StateMachine.intStateLastCycle) THEN
		CASE me.SubStateMachine.intState OF
			PTB_CmdState.cSUB_EMPTYWAITPAPERbusy:
				IF SIf.In.bolBeltExitSensor.intern THEN
					me.SubStateMachine.intStateNext := PTB_CmdState.cSUB_EMPTYWAITPAPERGONEbusy;
				END_IF
			PTB_CmdState.cSUB_EMPTYWAITPAPERGONEbusy:
				IF NOT SIf.In.bolBeltExitSensor.intern THEN
					SIf.Cur.uinPaperOnBelt := 0;
					cmd_STOP();
					me.SubStateMachine.intStateNext := PTB_CmdState.cSUB_EMPTYWAITDRIVESTOPED;
				END_IF
			PTB_CmdState.cSUB_EMPTYWAITDRIVESTOPED:
				IF (p_fbMotor^.CtrlCIf^.Job.intState = BASE_PLC.cSTA_STOP) THEN
					IF SIf.Par.bolAutoStackAfterEject THEN
						CIf.Job.intACmd := BASE_PLC.cCMD_DONE;
						CIf.Job.intMCmd := BASE_PLC.cCMD_DONE;
						me.StateMachine.intStateNext := PTB_CmdState.cSTA_STACKPAPERbusy;	
					ELSE	
						me.StateMachine.intStateNext := PTB_CmdState.cSTA_EJECTPAPER;	
					END_IF
				END_IF
		END_CASE
	END_IF


//--------------------------------------------------------------------------------------
// Exit action
	IF (me.StateMachine.intState<>me.StateMachine.intStateNext) THEN
		me.SubStateMachine.intState := BASE_PLC.cSTA_INITIALIZED;
	END_IF
END_METHOD

METHOD PROTECTED sta_ERROR : BOOL
// state implemetation
//--------------------------------------------------------------------------------------
// Entry action
	IF (me.StateMachine.intState<>me.StateMachine.intStateLastCycle) THEN
		me.StateMachine.intStateHistory := me.StateMachine.intStateLastCycle; // -> possibillity to go back to state before error
		me.StateMachine.intStateLastCycle := me.StateMachine.intState;
		pMotorCIf^.Job.intACmd := BASE_PLC.cCMD_OFF;		
	END_IF


//--------------------------------------------------------------------------------------
// Cyclic action
	IF (me.StateMachine.intState=me.StateMachine.intStateLastCycle) THEN
		
		;
		
		
		// State Change Condition
		IF (CIf.Job.bolAlmReset = TRUE) THEN
			me.StateMachine.intStateNext := cSTA_ERRORQuit;
		END_IF
	END_IF




//--------------------------------------------------------------------------------------
// Exit action
	IF (me.StateMachine.intState<>me.StateMachine.intStateNext) THEN
		;
	END_IF
END_METHOD

METHOD PROTECTED sta_ERRORQuit : BOOL
// state implemetation
//--------------------------------------------------------------------------------------
// Entry action
	IF (me.StateMachine.intState<>me.StateMachine.intStateLastCycle) THEN
		me.StateMachine.intStateLastCycle := me.StateMachine.intState;
		
	END_IF


//--------------------------------------------------------------------------------------
// Cyclic action
	IF (me.StateMachine.intState=me.StateMachine.intStateLastCycle) THEN
		
		;
		// evtl. wait time if reset of device is necessary and then decide to go to states or ERROR state
		IF (CIf.Job.bolAlmReset = TRUE) THEN
			CIf.Job.eMe_ActivAlmClass := E_AlmClass.NONE; // reset feedback channel for parent
			CIf.Job.bolAlmReset := FALSE;
		END_IF
		
		// State Change Condition
		IF (CIf.Job.bolAlmReset = FALSE) THEN
			IF (me.StateMachine.intStateHistory<=cSTA_PON) THEN
				me.StateMachine.intStateNext := cSTA_PONBusy;
			ELSIF(me.intCmd=cCMD_OFF) THEN
				me.StateMachine.intStateNext := cSTA_OFFBusy;
			ELSIF(me.intCmd=BASE_PLC.cCMD_RUN) THEN
				me.StateMachine.intStateNext := BASE_PLC.cSTA_RUNBusy;
			END_IF
		END_IF
	END_IF




//--------------------------------------------------------------------------------------
// Exit action
	IF (me.StateMachine.intState<>me.StateMachine.intStateNext) THEN
		;
	END_IF
END_METHOD

METHOD PROTECTED sta_OFF : BOOL
VAR_INPUT
END_VAR
// state implemetation
//--------------------------------------------------------------------------------------
// Entry action
	IF (me.StateMachine.intState<>me.StateMachine.intStateLastCycle) THEN
		me.StateMachine.intStateLastCycle := me.StateMachine.intState;
	END_IF


//--------------------------------------------------------------------------------------
// Cyclic action
	IF (me.StateMachine.intState=me.StateMachine.intStateLastCycle) THEN
		CASE me.intCmd OF
			BASE_PLC.cCMD_RUN:
				me.StateMachine.intStateNext := BASE_PLC.cSTA_RUNBusy;
			BASE_PLC.cCMD_STOP:
				me.StateMachine.intStateNext := BASE_PLC.cSTA_STOPBusy;
			PTB_CmdState.cCMD_EJECTPAPER:
				me.StateMachine.intStateNext := PTB_CmdState.cSTA_EJECTPAPERbusy;
			PTB_CmdState.cCMD_STACKPAPER:
				me.StateMachine.intStateNext := PTB_CmdState.cSTA_STACKPAPERbusy;
		END_CASE
	END_IF


//--------------------------------------------------------------------------------------
// Exit action
	IF (me.StateMachine.intState<>me.StateMachine.intStateNext) THEN
		;
	END_IF
END_METHOD

METHOD PROTECTED sta_OFFBusy : BOOL
VAR_INPUT
END_VAR
// state implemetation
//--------------------------------------------------------------------------------------
// Entry action
	IF (me.StateMachine.intState<>me.StateMachine.intStateLastCycle) THEN
		me.StateMachine.intStateLastCycle := me.StateMachine.intState;
		cmd_OFF();
	END_IF


//--------------------------------------------------------------------------------------
// Cyclic action
	IF (me.StateMachine.intState=me.StateMachine.intStateLastCycle) THEN

		// Set commandos not only in entry action because of possible errors or manual/auto changes
		cmd_OFF();

		IF p_fbMotor^.CtrlCIf^.Job.intState = BASE_PLC.cSTA_OFF 
		  AND CheckPumpState(BASE_PLC.cSTA_OFF) THEN
			me.StateMachine.intStateNext := BASE_PLC.cSTA_OFF;
		END_IF
	END_IF


//--------------------------------------------------------------------------------------
// Exit action
	IF (me.StateMachine.intState<>me.StateMachine.intStateNext) THEN
		;
	END_IF
END_METHOD

METHOD PROTECTED sta_PON : BOOL
VAR_INPUT
END_VAR
// state implemetation
//--------------------------------------------------------------------------------------
// Entry action
	IF (me.StateMachine.intState<>me.StateMachine.intStateLastCycle) THEN
		me.StateMachine.intStateLastCycle := me.StateMachine.intState;
		
	END_IF


//--------------------------------------------------------------------------------------
// Cyclic action
	IF (me.StateMachine.intState=me.StateMachine.intStateLastCycle) THEN
		;
	END_IF




//--------------------------------------------------------------------------------------
// Exit action
	IF (me.StateMachine.intState<>me.StateMachine.intStateNext) THEN
		;
	END_IF
END_METHOD

METHOD PROTECTED sta_RUN : Bool
VAR
	iDifference 		: INT;
END_VAR
// state implemetation
//--------------------------------------------------------------------------------------
// Entry action
	IF (me.StateMachine.intState<>me.StateMachine.intStateLastCycle) THEN
		me.StateMachine.intStateLastCycle := me.StateMachine.intState;
	END_IF


//--------------------------------------------------------------------------------------
// Cyclic action
	IF (me.StateMachine.intState = me.StateMachine.intStateLastCycle) THEN
		// The direction changed
		IF (SIf.Par.intDirection <> SIf.Cur.eActualDirection) THEN
			me.StateMachine.intStateNext := BASE_PLC.cSTA_RUNBusy;
		END_IF
		
		// The speed changed
		IF (SIf.Par.rBeltParam.uinBeltSpeed <> SIf.Cur.rBeltParam.uinBeltSpeed_mms) THEN
			me.StateMachine.intStateNext := BASE_PLC.cSTA_RUNBusy;
		END_IF
		
		IF  me.intCmd = BASE_PLC.cCMD_STOP THEN
			me.StateMachine.intStateNext := BASE_PLC.cSTA_STOPBusy;
		END_IF

		CASE SIf.Cfg.eMode OF
			E_PTB_MODE.ToDistance, 
			E_PTB_MODE.ToTime :
				IF me.StateMachine.udiTimeInState_ms > SIf.Cur.udiTimeToMove_ms THEN
					me.StateMachine.intStateNext := BASE_PLC.cSTA_STOPBusy;
				END_IF
			E_PTB_MODE.ToSensor:
				IF (SIf.In.bolBeltExitSensorPEdge.intern) THEN
					me.StateMachine.intStateNext := BASE_PLC.cSTA_STOPBusy;
				END_IF
		END_CASE
	END_IF


//--------------------------------------------------------------------------------------
// Exit action
	IF (me.StateMachine.intState<>me.StateMachine.intStateNext) THEN
		;
	END_IF
END_METHOD

METHOD PROTECTED sta_RUNBusy : BOOL
VAR_INPUT
END_VAR
// state implemetation
//--------------------------------------------------------------------------------------
// Entry action
	IF (me.StateMachine.intState<>me.StateMachine.intStateLastCycle) THEN
		me.StateMachine.intStateLastCycle := me.StateMachine.intState;
		
		CASE SIf.Cfg.eMode OF
			E_PTB_MODE.Endless,
			E_PTB_MODE.ToDistance,
			E_PTB_MODE.ToTime:
				cmd_RUN(sif.Par.rBeltParam.uinBeltSpeed);
			E_PTB_MODE.ToSensor:
				IF SIf.In.bolBeltExitSensorPEdge.intern THEN
					me.StateMachine.intStateNext := BASE_PLC.cSTA_STOPBusy;
				ELSE
					cmd_RUN(sif.Par.rBeltParam.uinBeltSpeed);
				END_IF
		END_CASE
	END_IF


//--------------------------------------------------------------------------------------
// Cyclic action
	IF (me.StateMachine.intState=me.StateMachine.intStateLastCycle) THEN
		IF (p_fbMotor^.CtrlCIf^.Job.intState = BASE_PLC.cSTA_RUN) 
		  AND (p_fbMotor^.CtrlSIf^.Cur.eDirection = arMotorDirection[SIf.Par.intDirection]) 
		  AND CheckPumpState(BASE_PLC.cSTA_RUN) THEN
			me.StateMachine.intStateNext := BASE_PLC.cSTA_RUN;
		END_IF

		IF me.intCmd = BASE_PLC.cCMD_STOP THEN
			me.StateMachine.intStateNext := BASE_PLC.cSTA_STOPBusy;
		END_IF
	END_IF


//--------------------------------------------------------------------------------------
// Exit action
	IF (me.StateMachine.intState<>me.StateMachine.intStateNext) THEN
		;
	END_IF
END_METHOD

METHOD PROTECTED sta_STACKPAPER : Bool
VAR
END_VAR
// state implemetation
//--------------------------------------------------------------------------------------
// Entry action
	IF (me.StateMachine.intState<>me.StateMachine.intStateLastCycle) THEN
		me.StateMachine.intStateLastCycle := me.StateMachine.intState;
	END_IF


//--------------------------------------------------------------------------------------
// Cyclic action
	IF (me.StateMachine.intState = me.StateMachine.intStateLastCycle) THEN
		CASE me.intCmd OF
			BASE_PLC.cCMD_RUN:
				me.StateMachine.intStateNext := BASE_PLC.cSTA_RUNBusy;
			BASE_PLC.cCMD_STOP:
				me.StateMachine.intStateNext := BASE_PLC.cSTA_STOPBusy;
			PTB_CmdState.cCMD_EJECTPAPER:
				me.StateMachine.intStateNext := PTB_CmdState.cSTA_EJECTPAPERbusy;
			PTB_CmdState.cCMD_STACKPAPER:
				me.StateMachine.intStateNext := PTB_CmdState.cSTA_STACKPAPERbusy;
		END_CASE
	END_IF


//--------------------------------------------------------------------------------------
// Exit action
	IF (me.StateMachine.intState<>me.StateMachine.intStateNext) THEN
		;
	END_IF
END_METHOD

METHOD PROTECTED sta_STACKPAPERbusy : BOOL
VAR_INPUT
END_VAR
// state implemetation
//--------------------------------------------------------------------------------------
// Entry action
	IF (me.StateMachine.intState<>me.StateMachine.intStateLastCycle) THEN
		me.StateMachine.intStateLastCycle := me.StateMachine.intState;

		me.SubStateMachine.intStateNext := PTB_CmdState.cSUB_WAITPAPER;
	END_IF


//--------------------------------------------------------------------------------------
// Cyclic action
	IF (me.StateMachine.intState=me.StateMachine.intStateLastCycle) THEN
		CASE me.SubStateMachine.intState OF
			PTB_CmdState.cSUB_WAITPAPER:
				IF SIf.In.bolBeltEntrySensor.intern THEN
					me.SubStateMachine.intStateNext := PTB_CmdState.cSUB_WAITPAPERGONE;
				ELSE
					CASE me.intCmd OF
						BASE_PLC.cCMD_RUN:
							me.StateMachine.intStateNext := BASE_PLC.cSTA_RUNBusy;
						BASE_PLC.cCMD_STOP:
							me.StateMachine.intStateNext := BASE_PLC.cSTA_STOPBusy;
						PTB_CmdState.cCMD_EJECTPAPER:
							me.StateMachine.intStateNext := PTB_CmdState.cSTA_EJECTPAPERbusy;
					END_CASE
				END_IF
			PTB_CmdState.cSUB_WAITPAPERGONE:
				IF NOT SIf.In.bolBeltEntrySensor.intern THEN
					SIf.Cur.uinPaperOnBelt := SIf.Cur.uinPaperOnBelt + 1;
					me.SubStateMachine.intStateNext := PTB_CmdState.cSUB_STARTSTACKDELAY;
				END_IF
			PTB_CmdState.cSUB_STARTSTACKDELAY:
				IF me.SubStateMachine.udiTimeInState_ms > SIf.Par.udiStackDelayTime_ms THEN
					IF SIf.Cur.uinPaperOnBelt >= SIf.Par.uinPaperStackHight THEN
						me.StateMachine.intStateNext := PTB_CmdState.cSTA_EJECTPAPERbusy;
					ELSE
						me.SubStateMachine.intStateNext := PTB_CmdState.cSUB_PAPERDISTANCEstart;
					END_IF
				END_IF
			PTB_CmdState.cSUB_PAPERDISTANCEstart:
				cmd_RUN(sif.Par.rBeltParam.uinStackSpeed);
				me.SubStateMachine.intStateNext := PTB_CmdState.cSUB_PAPERDISTANCEbusy;
			PTB_CmdState.cSUB_PAPERDISTANCEbusy:
				IF me.SubStateMachine.udiTimeInState_ms > SIf.Cur.udiTimeToMove_ms THEN
					cmd_STOP();
					me.SubStateMachine.intStateNext := PTB_CmdState.cSUB_PAPERDISTANCESTOPbusy;
				END_IF
			PTB_CmdState.cSUB_PAPERDISTANCESTOPbusy:
				IF p_fbMotor^.CtrlCIf^.Job.intState = BASE_PLC.cSTA_STOP THEN
					IF SIf.Par.bolAutoEjectAfterStack THEN
						me.StateMachine.intStateNext := PTB_CmdState.cSTA_EJECTPAPERbusy;
					ELSE
						me.StateMachine.intStateNext := PTB_CmdState.cSTA_STACKPAPER;
					END_IF
				END_IF
		END_CASE
	END_IF


//--------------------------------------------------------------------------------------
// Exit action
	IF (me.StateMachine.intState<>me.StateMachine.intStateNext) THEN
		CIf.Job.intACmd := BASE_PLC.cCMD_DONE;
		CIf.Job.intMCmd := BASE_PLC.cCMD_DONE;
		me.SubStateMachine.intState := BASE_PLC.cSTA_INITIALIZED;
	END_IF
END_METHOD

METHOD PROTECTED sta_STOP : BOOL
VAR_INPUT
END_VAR
// state implemetation
//--------------------------------------------------------------------------------------
// Entry action
	IF (me.StateMachine.intState<>me.StateMachine.intStateLastCycle) THEN
		me.StateMachine.intStateLastCycle := me.StateMachine.intState;
	END_IF


//--------------------------------------------------------------------------------------
// Cyclic action
	IF (me.StateMachine.intState=me.StateMachine.intStateLastCycle) THEN
		CASE me.intCmd OF
			BASE_PLC.cCMD_RUN:
				me.StateMachine.intStateNext := BASE_PLC.cSTA_RUNBusy;
			BASE_PLC.cCMD_STOP:
				me.StateMachine.intStateNext := BASE_PLC.cSTA_STOPBusy;
			PTB_CmdState.cCMD_EJECTPAPER:
				me.StateMachine.intStateNext := PTB_CmdState.cSTA_EJECTPAPERbusy;
			PTB_CmdState.cCMD_STACKPAPER:
				me.StateMachine.intStateNext := PTB_CmdState.cSTA_STACKPAPERbusy;
		END_CASE

		IF    (SIf.Cfg.eMode = E_PTB_MODE.ToSensor) 
		  AND (SIf.In.bolBeltExitSensorNEdge.intern) THEN
			me.StateMachine.intStateNext := BASE_PLC.cSTA_RUNBusy;
		END_IF
	END_IF


//--------------------------------------------------------------------------------------
// Exit action
	IF (me.StateMachine.intState<>me.StateMachine.intStateNext) THEN
		;
	END_IF
END_METHOD

METHOD PROTECTED sta_STOPBusy : BOOL
VAR_INPUT
END_VAR
// state implemetation
//--------------------------------------------------------------------------------------
// Entry action
	IF (me.StateMachine.intState<>me.StateMachine.intStateLastCycle) THEN
		me.StateMachine.intStateLastCycle := me.StateMachine.intState;
		cmd_STOP();
	END_IF


//--------------------------------------------------------------------------------------
// Cyclic action
	IF (me.StateMachine.intState=me.StateMachine.intStateLastCycle) THEN
		IF p_fbMotor^.CtrlCIf^.Job.intState = BASE_PLC.cSTA_STOP  THEN
			me.StateMachine.intStateNext := BASE_PLC.cSTA_STOP;
		END_IF
	END_IF


//--------------------------------------------------------------------------------------
// Exit action
	IF (me.StateMachine.intState<>me.StateMachine.intStateNext) THEN
		;
	END_IF
END_METHOD

METHOD PROTECTED StateMachine : BOOL
SUPER^.StateMachine();

// main statemachine of base controller
CASE me.StateMachine.intState OF
    BASE_PLC.cSTA_RUN: 
        THIS^.sta_RUN();
    BASE_PLC.cSTA_RUNBusy: 
        THIS^.sta_RUNBusy();
    BASE_PLC.cSTA_STOP: 
        THIS^.sta_STOP();
    BASE_PLC.cSTA_STOPBusy: 
        THIS^.sta_STOPBusy();
	PTB_CmdState.cSTA_EJECTPAPERbusy:
		THIS^.sta_EJECTPAPERbusy();
	PTB_CmdState.cSTA_EJECTPAPER:
		THIS^.sta_EJECTPAPER();
	PTB_CmdState.cSTA_STACKPAPER:
		THIS^.sta_STACKPAPER();
	PTB_CmdState.cSTA_STACKPAPERbusy:
		THIS^.sta_STACKPAPERbusy();
END_CASE;
END_METHOD

PROPERTY PUBLIC VacuumPump :  POINTER TO FB_VPC
GET
VacuumPump := p_fbPump;
END_GET
SET
p_fbPump := VacuumPump;
END_SET
END_PROPERTY

END_FUNCTION_BLOCK

// POUs/Controller/Lvl2/PBC [Paper Buffer Controller]/helper/cycle_Pbc
FUNCTION cycle_Pbc : BOOL
VAR_INPUT
	pPbc: POINTER TO T_PBC;
END_VAR

pPbc^.ctrl.fbPbc_PtbDeStacker_Umc.In_uinStatus 				:= pPbc^.io.In_uinPtbDeStacker_Umc_Status;
pPbc^.ctrl.fbPbc_PtbDeStacker_Umc.In_intMotorActualSpeed 	:= pPbc^.io.In_uinPtbDeStacker_Umc_ActualSpeed;
pPbc^.ctrl.fbPbc_PtbDeStacker_Umc.In_uinMotorSetSpeed 		:= pPbc^.io.In_uinPtbDeStacker_Umc_SetSpeed;
pPbc^.ctrl.fbPbc_PtbDeStacker_Umc.In_uinIOData				:= pPbc^.io.In_uinPtbDeStacker_Umc_IOData1;
pPbc^.ctrl.fbPbc_PtbDeStacker_Umc.In_uinECATState 			:= pPbc^.io.In_uinPtbDeStacker_Umc_ECatState;
pPbc^.ctrl.fbPbc_PtbDeStacker_Umc.In_strNetId 				:= pPbc^.io.In_strPtbDeStacker_Umc_ECatNetId;
pPbc^.ctrl.fbPbc_PtbDeStacker_Umc.In_uintPort 				:= pPbc^.io.In_uinPtbDeStacker_Umc_ECatPort;
pPbc^.ctrl.fbPbc_PtbDeStacker_Umc();
pPbc^.io.Out_uinPtbDeStacker_Umc_SetSpeed	 				:= pPbc^.ctrl.fbPbc_PtbDeStacker_Umc.Out_uinSpeedSetpoint;
pPbc^.io.Out_uinPtbDeStacker_Umc_Control 					:= pPbc^.ctrl.fbPbc_PtbDeStacker_Umc.Out_uinControl;

pPbc^.ctrl.fbPbc_PtbDeStacker();

pPbc^.ctrl.fbPbc_PtbBelt_Umc.In_uinStatus 					:= pPbc^.io.In_uinPtbBelt_Umc_Status;
pPbc^.ctrl.fbPbc_PtbBelt_Umc.In_intMotorActualSpeed 		:= pPbc^.io.In_uinPtbBelt_Umc_ActualSpeed;
pPbc^.ctrl.fbPbc_PtbBelt_Umc.In_uinMotorSetSpeed 			:= pPbc^.io.In_uinPtbBelt_Umc_SetSpeed;
pPbc^.ctrl.fbPbc_PtbBelt_Umc.In_uinIOData					:= pPbc^.io.In_uinPtbBelt_Umc_IOData1;
pPbc^.ctrl.fbPbc_PtbBelt_Umc.In_uinECATState 				:= pPbc^.io.In_uinPtbBelt_Umc_ECatState;
pPbc^.ctrl.fbPbc_PtbBelt_Umc.In_strNetId 					:= pPbc^.io.In_strPtbBelt_Umc_ECatNetId;
pPbc^.ctrl.fbPbc_PtbBelt_Umc.In_uintPort 					:= pPbc^.io.In_uinPtbBelt_Umc_ECatPort;
pPbc^.ctrl.fbPbc_PtbBelt_Umc();
pPbc^.io.Out_uinPtbBelt_Umc_SetSpeed 						:= pPbc^.ctrl.fbPbc_PtbBelt_Umc.Out_uinSpeedSetpoint;
pPbc^.io.Out_uinPtbBelt_Umc_Control 						:= pPbc^.ctrl.fbPbc_PtbBelt_Umc.Out_uinControl;

pPbc^.ctrl.fbPbc_PtbBelt_Vpc.In_bolPumpOk 					:= pPbc^.io.In_bolPtbBelt_Vpc_PumpOk;
pPbc^.ctrl.fbPbc_PtbBelt_Vpc.In_bolVacuumOk 				:= pPbc^.io.In_bolPtbBelt_Vpc_VacuumSensor;
pPbc^.ctrl.fbPbc_PtbBelt_Vpc();
pPbc^.io.Out_bolPtbBelt_Vpc_PumpOn 							:= pPbc^.ctrl.fbPbc_PtbBelt_Vpc.Out_bolVaccumPumpOn;

pPbc^.ctrl.fbPbc_PtbBelt();

pPbc^.ctrl.fbPbc.In_bolCapacityReached 						:= pPbc^.io.In_bolInputSensor;
pPbc^.ctrl.fbPbc.In_bolPaperAvailableEntry 					:= pPbc^.io.In_bolCapacitySensor;
pPbc^.ctrl.fbPbc.In_bolPaperAvailableExit 					:= pPbc^.io.In_bolOutputSensor;
pPbc^.ctrl.fbPbc.In_bolDoublePaperDetection 				:= pPbc^.io.In_bolDoublePaperSensor;
pPbc^.ctrl.fbPbc.In_bolTurnTableMiddleSensor 				:= pPbc^.io.In_bolPts_PaperSensor;
pPbc^.ctrl.fbPbc.In_bolAirPressorOk 						:= pPbc^.io.In_bolAirPressureOk;
pPbc^.ctrl.fbPbc();
pPbc^.io.Out_bolAirPressureOn 								:= pPbc^.ctrl.fbPbc.Out_bolAirOn;

END_FUNCTION

// POUs/Controller/Lvl2/PBC [Paper Buffer Controller]/helper/init_Pbc
FUNCTION init_Pbc : BOOL
VAR_INPUT
	pPbc: POINTER TO T_PBC;
	/// instance array of all controller instances
	pCtrlInst: POINTER TO fb_CtrlBase;
	/// common interface array of all controllers (main use for PLC)
	pCtrlCIf: POINTER TO T_Ctrl_CIf;
END_VAR

pPbc^.ctrl.fbPbc_PtbDeStacker_Umc.iniAllCtrlArrays(pCtrlInst,pCtrlCIf,pPbc^.id.Pbc_PtbDeStacker_Umc); // init and entry fb_instance in global fb pointer array
pPbc^.ctrl.fbPbc_PtbDeStacker.iniAllCtrlArrays(pCtrlInst,pCtrlCIf,pPbc^.id.Pbc_PtbDeStacker); // init and entry fb_instance in global fb pointer array
pPbc^.ctrl.fbPbc_PtbDeStacker.Drive := ADR(pPbc^.ctrl.fbPbc_PtbDeStacker_Umc);

pPbc^.ctrl.fbPbc_PtbBelt_Umc.iniAllCtrlArrays(pCtrlInst,pCtrlCIf,pPbc^.id.Pbc_PtbBelt_Umc); // init and entry fb_instance in global fb pointer array
pPbc^.ctrl.fbPbc_PtbBelt_Vpc.iniAllCtrlArrays(pCtrlInst,pCtrlCIf,pPbc^.id.Pbc_PtbBelt_Vpc); // init and entry fb_instance in global fb pointer array
pPbc^.ctrl.fbPbc_PtbBelt.iniAllCtrlArrays(pCtrlInst,pCtrlCIf,pPbc^.id.Pbc_PtbBelt); // init and entry fb_instance in global fb pointer array
pPbc^.ctrl.fbPbc_PtbBelt.Drive := ADR(pPbc^.ctrl.fbPbc_PtbBelt_Umc);
pPbc^.ctrl.fbPbc_PtbBelt.VacuumPump := ADR(pPbc^.ctrl.fbPbc_PtbBelt_Vpc);

pPbc^.ctrl.fbPbc.iniAllCtrlArrays(pCtrlInst,pCtrlCIf,pPbc^.id.Pbc); 		 // init and entry fb_instance in global fb pointer array
pPbc^.ctrl.fbPbc.DeStacker := ADR(pPbc^.ctrl.fbPbc_PtbDeStacker);
pPbc^.ctrl.fbPbc.Belt := ADR(pPbc^.ctrl.fbPbc_PtbBelt);

END_FUNCTION

// POUs/Controller/Lvl2/PBC [Paper Buffer Controller]/FB_PBC
FUNCTION_BLOCK FB_PBC EXTENDS FB_CtrlBase
VAR_INPUT
	In_bolPaperAvailableExit: BOOL;
	In_bolPaperAvailableEntry: BOOL;
	In_bolCapacityReached: BOOL;
	In_bolDoublePaperDetection: BOOL;
	In_bolTurnTableMiddleSensor: BOOL;
	In_bolAirPressorOk: BOOL;
END_VAR
VAR_OUTPUT
	Out_bolAirOn: BOOL;
END_VAR
VAR
	/// Specific interface struct for public access
	/// -------------------------------------------------------
	SIf: T_Ctrl_SIf_PBC;
	///Sub Controller Pointer
	/// -------------------------------------------------------
	p_fbDeStacker: POINTER TO FB_PTB;
	pDeStackerCIf: POINTER TO BASE_PLC.T_Ctrl_CIf;
	p_fbBelt: POINTER TO FB_PTB;
	pBeltCIf: POINTER TO BASE_PLC.T_Ctrl_CIf;
	/// Other localy used variables
	/// -------------------------------------------------------
	m_uinPaperHight_mm: UINT := 460;
	m_uinPaperWidth_mm: UINT := 320;
	m_intRetry: INT := 0;
	udiBufferEmptyTimer_ms: UDINT;
END_VAR
VAR CONSTANT
	cPAPERPOSITION_TOLERANCE_mm: UINT := 200;
END_VAR

(*__________________________________________________________________________________________________
¦	
¦	Vistaprint Schweiz GmbH
¦	CH - 8401 Winterthur
¦
¦	www.vistaprint.ch - info@vistaprint.ch
¦___________________________________________________________________________________________________

Function desription:
Destacker/Buffer implementation. 


History:
Version		Date			Author		Comment
---------------------------------------------------------------------------------------------------
0.00.1		09.07.2013		PC			Start history
0.00.2		05.02.2015		RE			React on StopReleaseItems flag to stop destacking
0.00.3		06.02.2015		RE			Bug fix StopReleaseItems, fixed some comments
___________________________________________________________________________________________________*)


SUPER^();

{attribute 'object_name' := 'Always'}
METHOD PROTECTED Always : BOOL
VAR
	pItem: POINTER TO T_IdBase_DCH;
	bResult: BOOL;
END_VAR
SUPER^.Always();

// ----------------------------------------------------------------------------------
// cyclic actions outside of statemachine
IF (me.StateMachine.intState<>cSTA_SINGLE_ANSWER) THEN
	
	// check if DeStacker is empty
	IF NOT SIf.In.bolPaperAvailableEntry.intern AND NOT SIf.In.bolPaperAvailableExit.intern THEN
		udiBufferEmptyTimer_ms := udiBufferEmptyTimer_ms + me.FUBInfo.udiSample_ms;
		IF udiBufferEmptyTimer_ms > 3000 THEN
			SIf.Cur.intPaperInBufferCount := 0;
		END_IF
	ELSE
		udiBufferEmptyTimer_ms := 0;
		SIf.Cur.intPaperInBufferCount := -1;
	END_IF

END_IF

// ----------------------------------------------------------------------------------
// Conditions Always
IF (((me.Alarm.eActivAlmClass=E_AlmClass.EOFF) OR (me.Alarm.eActivAlmClass=E_AlmClass.OFF) OR (me.intCmd=cCMD_OFF) OR (me.intCmd=BASE_PLC.cCMD_EOFF))
		 AND (me.StateMachine.intState<>cSTA_ERROR) AND (me.StateMachine.intState<>cSTA_ERRORQuit) AND
		(me.StateMachine.intState<>cSTA_OFF) AND (me.StateMachine.intState<>cSTA_OFFBusy)) THEN
	// alarm evt EOFF, OFF or cmd off
	me.StateMachine.intStateNext := cSTA_OFFBusy;
END_IF
END_METHOD

PROPERTY Belt : POINTER TO FB_PTB
GET
Belt := p_fbBelt;
END_GET
SET
p_fbBelt := Belt;
END_SET
END_PROPERTY

{attribute 'object_name' := 'CountPaper'}
METHOD PROTECTED CountPaper : UINT
END_METHOD

{attribute 'object_name' := 'CtrlInit'}
METHOD CtrlInit : BOOL
VAR
	pBccSIf: POINTER TO T_Ctrl_SIf_BCC;
END_VAR
SUPER^.CtrlInit();

pDeStackerCIf 	:= AddChild(p_fbDeStacker^);
pBeltCIf 		:= AddChild(p_fbBelt^);
END_METHOD

PROPERTY CtrlSIf : POINTER TO T_Ctrl_SIf_PBC
GET
CtrlSIf := ADR(SIf);
END_GET
END_PROPERTY

PROPERTY DeStacker : POINTER TO FB_PTB
GET
DeStacker := p_fbDeStacker;
END_GET
SET
p_fbDeStacker := DeStacker;
END_SET
END_PROPERTY

{attribute 'object_name' := 'FB_init'}
METHOD FB_init : BOOL
VAR_INPUT
	/// if TRUE, the retain variables are initialized (warm start / cold start)
	bInitRetains: BOOL;
	/// if TRUE, the instance afterwards gets moved into the copy code (online change)
	bInCopyCode: BOOL;
END_VAR
VAR
	iIdx: UINT;
	iLength: UINT;
END_VAR
//------------------------------------------------------------------------------------------------------------------------
// to manually change in new FUB implementation!!!
// define valid commands for this controller
iLength := SIZEOF(CIf.Job.aCmdList)/SIZEOF(CIf.Job.aCmdList[0]);
iIdx := 0;

WHILE (iIdx < iLength) AND (CIf.Job.aCmdList[iIdx].intCmd <> cCMD_INITIALIZED) DO
	iIdx := iIdx + 1; 
END_WHILE

IF (iIdx < iLength) THEN
// Add configuration of own comands	
	CIf.Job.aCmdList[iIdx].intCmd := BASE_PLC.cCMD_RUN;
	CIf.Job.aCmdList[iIdx].strName := 'RUN'; 
	CIf.Job.aCmdList[iIdx].bolAvailable := TRUE;
	iIdx := iIdx + 1;
	CIf.Job.aCmdList[iIdx].intCmd := BASE_PLC.cCMD_STOP;
	CIf.Job.aCmdList[iIdx].strName := 'STOP'; 
	CIf.Job.aCmdList[iIdx].bolAvailable := TRUE;
	iIdx := iIdx + 1;
	CIf.Job.aCmdList[iIdx].intCmd := PBC_CmdState.cCMD_SINGLE;
	CIf.Job.aCmdList[iIdx].strName := 'SINGLE'; 
	CIf.Job.aCmdList[iIdx].bolAvailable := TRUE;
ELSE
	// Error if the aCmdList Array is to small
END_IF

// set name of class/typ
CIf.Info.strType := 'FB_PBC';  
CIf.Info.strFullName := 'Paper Buffer Controller';

// set alarm class
SIf.Alm[E_ALM_PBC.BufferEmpty].eAlmClass := Base_PLC.E_AlmClass.WARNING;
SIf.Alm[E_ALM_PBC.BufferEmpty].strText := 'Buffer is Empty'; 
SIf.Alm[E_ALM_PBC.BufferFull].eAlmClass := E_AlmClass.TSTOP;
SIf.Alm[E_ALM_PBC.BufferFull].strText := 'Buffer reached capacity limit';
SIf.Alm[E_ALM_PBC.PaperTransport].eAlmClass := E_AlmClass.TSTOP;
SIf.Alm[E_ALM_PBC.PaperTransport].strText := 'Possible Paper Jam';
SIf.Alm[E_ALM_PBC.DoublePaperError].eAlmClass := E_AlmClass.TSTOP;
SIf.Alm[E_ALM_PBC.DoublePaperError].strText := 'Double paper detected';
SIf.Alm[E_ALM_PBC.DataChannelBufferFull].eAlmClass := E_AlmClass.WARNING;
SIf.Alm[E_ALM_PBC.DataChannelBufferFull].strText := 'Data Channel buffer is full';
SIf.Alm[E_ALM_PBC.DataChannelSend].eAlmClass := E_AlmClass.WARNING;
SIf.Alm[E_ALM_PBC.DataChannelSend].strText := 'Data Channel item could not be sent';
SIf.Alm[E_ALM_PBC.PaperInject].eAlmClass := E_AlmClass.TSTOP;
SIf.Alm[E_ALM_PBC.PaperInject].strText := 'Paper is not transported to the front';
SIf.Alm[E_ALM_PBC.PaperInjectRetry].eAlmClass := E_AlmClass.WARNING;
SIf.Alm[E_ALM_PBC.PaperInjectRetry].strText := 'Paper transport retry';
SIf.Alm[E_ALM_PBC.DoNotReleaseItems].eAlmClass := E_AlmClass.INFO;
SIf.Alm[E_ALM_PBC.DoNotReleaseItems].strText := 'Currently not releasing items because in manual mode';
SIf.Alm[E_ALM_PBC.DoublePaperWarning].eAlmClass := E_AlmClass.WARNING;
SIf.Alm[E_ALM_PBC.DoublePaperWarning].strText := 'Double paper detected';

//*******************************************************************************
// initial values
//*******************************************************************************

// software configuration
CIf.SwCfg.bolExist := TRUE;
CIf.SwCfg.bolEnable := TRUE;
CIf.SwCfg.bolSimulation := FALSE;

// Configuration
SIf.Cfg.bolUseTurnTableSensorForEject 		:= TRUE;
SIf.Cfg.bolEnableDataChannel		  		:= FALSE;
SIf.Cfg.bolGranulatAirPressureUnitAvailable := FALSE;
SIf.Cfg.bolEnableSaberStopDeStack 			:= TRUE;

// parameter
SIf.Par.bolAutomaticMode := FALSE;
SIf.Par.bolStopReleaseItems := FALSE;
SIf.Par.udiPaperTransportTime := 3000;
SIf.Par.udiSheetToEject := 0;
SIf.Par.udiSheetToSheetTime := 22800;
SIf.Par.udiManualSheetToSheetTime_ms := 22800;
SIf.Par.udiPaperInjectRetryPauseTime_ms := 400;
SIf.Par.udiPaperInjectRetries := 3;
SIf.Par.udiDoublePaperDebounceTime_ms := 500;
SIf.Par.bolEnableDoublePaperDetection := FALSE;
SIf.Par.udiSimPaperTransportTime := SIf.Par.udiPaperTransportTime / 2;
SIf.Par.udiSimPaperToPaperTransportTime := SIf.Par.udiPaperTransportTime / 20;
END_METHOD

{attribute 'object_name' := 'getCmdState'}
METHOD PROTECTED getCmdState : STRING
VAR_INPUT
	intCmdState: INT;
	bolState: BOOL;
END_VAR
getCmdState := SUPER^.getCmdState(intCmdState:=intCmdState,bolState:=bolState); // get global/base defined cmds/states

